LIN {X 0,Y 227.933,Z 465.716,A -85,B 0,C 180,E1 -20092.329,E2 -20092.329} C_VEL
LIN {X 0,Y 227.945,Z 465.715,A -85,B 0,C 180,E1 -20096.602,E2 -20096.602} C_VEL
LIN {X 0,Y 227.902,Z 465.721,A -85,B 0,C 180,E1 -20100.292,E2 -20100.292} C_VEL
LIN {X 0,Y 227.747,Z 465.74,A -85,B 0,C 180,E1 -20103.742,E2 -20103.742} C_VEL
LIN {X 0,Y 227.512,Z 465.771,A -85,B 0,C 180,E1 -20106.566,E2 -20106.566} C_VEL
LIN {X 0,Y 227.279,Z 465.972,A -85,B 0,C 180,E1 -20109.146,E2 -20109.146} C_VEL
LIN {X 0,Y 231.965,Z 479.924,A -85,B 0,C 180,E1 -20110.648,E2 -20110.648} C_VEL
LIN {X 0,Y 235.68,Z 494.545,A -85,B 0,C 180,E1 -20112.428,E2 -20112.428} C_VEL
LIN {X 0,Y 238.49,Z 507.946,A -85,B 0,C 180,E1 -20114.33,E2 -20114.33} C_VEL
LIN {X 0,Y 238.944,Z 511.073,A -85,B 0,C 180,E1 -20114.799,E2 -20114.799} C_VEL
LIN {X 0,Y 236.811,Z 523.709,A -85,B 0,C 180,E1 -20116.662,E2 -20116.662} C_VEL
LIN {X 0,Y 234.596,Z 535.4,A -85,B 0,C 180,E1 -20118.77,E2 -20118.77} C_VEL
LIN {X 0,Y 232.314,Z 547.285,A -85,B 0,C 180,E1 -20121.409,E2 -20121.409} C_VEL
LIN {X 0,Y 230.404,Z 556.987,A -85,B 0,C 180,E1 -20124.042,E2 -20124.042} C_VEL
LIN {X 0,Y 228.727,Z 565.771,A -85,B 0,C 180,E1 -20126.948,E2 -20126.948} C_VEL
LIN {X 0,Y 227.575,Z 572.918,A -85,B 0,C 180,E1 -20129.847,E2 -20129.847} C_VEL
LIN {X 0,Y 226.553,Z 579.643,A -85,B 0,C 180,E1 -20133.269,E2 -20133.269} C_VEL
LIN {X 0,Y 225.996,Z 584.123,A -85,B 0,C 180,E1 -20136.154,E2 -20136.154} C_VEL
LIN {X 0,Y 225.683,Z 587.632,A -85,B 0,C 180,E1 -20139.101,E2 -20139.101} C_VEL
LIN {X 0,Y 225.632,Z 589.987,A -85,B 0,C 180,E1 -20141.851,E2 -20141.851} C_VEL
LIN {X 0,Y 226.022,Z 591.964,A -85,B 0,C 180,E1 -20145.596,E2 -20145.596} C_VEL
LIN {X 0,Y 226.859,Z 592.527,A -85,B 0,C 180,E1 -20149.287,E2 -20149.287} C_VEL
LIN {X 0,Y 228.331,Z 591.732,A -85,B 0,C 180,E1 -20152.927,E2 -20152.927} C_VEL
LIN {X 0,Y 230.472,Z 589.612,A -85,B 0,C 180,E1 -20156.503,E2 -20156.503} C_VEL
LIN {X 0,Y 233.31,Z 586.131,A -85,B 0,C 180,E1 -20160,E2 -20160} C_VEL
LIN {X 0,Y 237.001,Z 581.247,A -85,B 0,C 180,E1 -20163.4,E2 -20163.4} C_VEL
LIN {X 0,Y 241.37,Z 574.833,A -85,B 0,C 180,E1 -20166.688,E2 -20166.688} C_VEL
LIN {X 0,Y 245.945,Z 567.842,A -85,B 0,C 180,E1 -20169.457,E2 -20169.457} C_VEL
LIN {X 0,Y 251.115,Z 559.281,A -85,B 0,C 180,E1 -20172.117,E2 -20172.117} C_VEL
LIN {X 0,Y 256.753,Z 549.023,A -85,B 0,C 180,E1 -20174.666,E2 -20174.666} C_VEL
LIN {X 0,Y 262.048,Z 538.351,A -85,B 0,C 180,E1 -20176.757,E2 -20176.757} C_VEL
LIN {X 0,Y 262.469,Z 536.8,A -85,B 0,C 180,E1 -20177.13,E2 -20177.13} C_VEL
LIN {X 0,Y 262.228,Z 531.504,A -85,B 0,C 180,E1 -20179.059,E2 -20179.059} C_VEL
LIN {X 0,Y 261.499,Z 526.204,A -85,B 0,C 180,E1 -20181.251,E2 -20181.251} C_VEL
LIN {X 0,Y 260.237,Z 521.055,A -85,B 0,C 180,E1 -20183.897,E2 -20183.897} C_VEL
LIN {X 0,Y 259.201,Z 518.357,A -85,B 0,C 180,E1 -20185.71,E2 -20185.71} C_VEL
LIN {X 0,Y 258.204,Z 516.399,A -85,B 0,C 180,E1 -20187.563,E2 -20187.563} C_VEL
LIN {X 0,Y 257.317,Z 514.957,A -85,B 0,C 180,E1 -20189.447,E2 -20189.447} C_VEL
LIN {X 0,Y 256.6,Z 513.704,A -85,B 0,C 180,E1 -20191.892,E2 -20191.892} C_VEL
LIN {X 0,Y 256.346,Z 513.407,A -85,B 0,C 180,E1 -20193.252,E2 -20193.252} C_VEL
LIN {X 0,Y 256.04,Z 513.801,A -85,B 0,C 180,E1 -20195.199,E2 -20195.199} C_VEL
LIN {X 0,Y 256.535,Z 515.763,A -85,B 0,C 180,E1 -20199.058,E2 -20199.058} C_VEL
LIN {X 0,Y 257.505,Z 521.048,A -85,B 0,C 180,E1 -20203.025,E2 -20203.025} C_VEL
LIN {X 0,Y 258.198,Z 524.969,A -85,B 0,C 180,E1 -20205.048,E2 -20205.048} C_VEL
LIN {X 0,Y 258.639,Z 529.116,A -85,B 0,C 180,E1 -20206.725,E2 -20206.725} C_VEL
LIN {X 0,Y 258.68,Z 537.141,A -85,B 0,C 180,E1 -20209.305,E2 -20209.305} C_VEL
LIN {X 0,Y 258.66,Z 537.501,A -85,B 0,C 180,E1 -20209.412,E2 -20209.412} C_VEL
LIN {X 0,Y 257.951,Z 541.489,A -85,B 0,C 180,E1 -20210.377,E2 -20210.377} C_VEL
LIN {X 0,Y 256.451,Z 545.94,A -85,B 0,C 180,E1 -20211.202,E2 -20211.202} C_VEL
LIN {X 0,Y 251.158,Z 557.863,A -85,B 0,C 180,E1 -20213.305,E2 -20213.305} C_VEL
LIN {X 0,Y 250.114,Z 560.562,A -85,B 0,C 180,E1 -20213.936,E2 -20213.936} C_VEL
LIN {X 0,Y 247.79,Z 566.678,A -85,B 0,C 180,E1 -20215.442,E2 -20215.442} C_VEL
LIN {X 0,Y 242.545,Z 575.941,A -85,B 0,C 180,E1 -20217.585,E2 -20217.585} C_VEL
LIN {X 0,Y 237.104,Z 585.099,A -85,B 0,C 180,E1 -20220.233,E2 -20220.233} C_VEL
LIN {X 0,Y 233.036,Z 591.862,A -85,B 0,C 180,E1 -20222.619,E2 -20222.619} C_VEL
LIN {X 0,Y 228.918,Z 598.493,A -85,B 0,C 180,E1 -20225.515,E2 -20225.515} C_VEL
LIN {X 0,Y 225.038,Z 604.726,A -85,B 0,C 180,E1 -20228.953,E2 -20228.953} C_VEL
LIN {X 0,Y 222.166,Z 609.536,A -85,B 0,C 180,E1 -20232.511,E2 -20232.511} C_VEL
LIN {X 0,Y 220.591,Z 612.29,A -85,B 0,C 180,E1 -20235.234,E2 -20235.234} C_VEL
LIN {X 0,Y 219.223,Z 614.884,A -85,B 0,C 180,E1 -20238.91,E2 -20238.91} C_VEL
LIN {X 0,Y 218.689,Z 616.234,A -85,B 0,C 180,E1 -20242.614,E2 -20242.614} C_VEL
LIN {X 0,Y 218.848,Z 616.308,A -85,B 0,C 180,E1 -20246.318,E2 -20246.318} C_VEL
LIN {X 0,Y 219.08,Z 615.033,A -85,B 0,C 180,E1 -20250,E2 -20250} C_VEL
LIN {X 0,Y 218.976,Z 612.273,A -85,B 0,C 180,E1 -20253.68,E2 -20253.68} C_VEL
LIN {X 0,Y 219.06,Z 609.777,A -85,B 0,C 180,E1 -20255.981,E2 -20255.981} C_VEL
LIN {X 0,Y 219.178,Z 605.128,A -85,B 0,C 180,E1 -20259.226,E2 -20259.226} C_VEL
LIN {X 0,Y 219.659,Z 600.055,A -85,B 0,C 180,E1 -20262.003,E2 -20262.003} C_VEL
LIN {X 0,Y 220.616,Z 592.746,A -85,B 0,C 180,E1 -20265.237,E2 -20265.237} C_VEL
LIN {X 0,Y 222.212,Z 583.656,A -85,B 0,C 180,E1 -20268.437,E2 -20268.437} C_VEL
LIN {X 0,Y 224.07,Z 574.212,A -85,B 0,C 180,E1 -20271.143,E2 -20271.143} C_VEL
LIN {X 0,Y 226.416,Z 562.842,A -85,B 0,C 180,E1 -20273.798,E2 -20273.798} C_VEL
LIN {X 0,Y 228.937,Z 550.545,A -85,B 0,C 180,E1 -20276.121,E2 -20276.121} C_VEL
LIN {X 0,Y 228.849,Z 545.123,A -85,B 0,C 180,E1 -20277.052,E2 -20277.052} C_VEL
LIN {X 0,Y 227.742,Z 532.027,A -85,B 0,C 180,E1 -20279.08,E2 -20279.08} C_VEL
LIN {X 0,Y 226.226,Z 517.932,A -85,B 0,C 180,E1 -20280.909,E2 -20280.909} C_VEL
LIN {X 0,Y 224.184,Z 502.881,A -85,B 0,C 180,E1 -20282.529,E2 -20282.529} C_VEL
LIN {X 0,Y 221.762,Z 487.259,A -85,B 0,C 180,E1 -20283.908,E2 -20283.908} C_VEL
LIN {X 0,Y 222.836,Z 482.859,A -85,B 0,C 180,E1 -20287.957,E2 -20287.957} C_VEL
LIN {X 0,Y 223.128,Z 479.233,A -85,B 0,C 180,E1 -20291.41,E2 -20291.41} C_VEL
LIN {X 0,Y 222.752,Z 476.696,A -85,B 0,C 180,E1 -20293.956,E2 -20293.956} C_VEL
LIN {X 0,Y 221.937,Z 472.506,A -85,B 0,C 180,E1 -20298.318,E2 -20298.318} C_VEL
LIN {X 0,Y 221.216,Z 468.39,A -85,B 0,C 180,E1 -20302.87,E2 -20302.87} C_VEL
LIN {X 0,Y 220.928,Z 466.591,A -85,B 0,C 180,E1 -20305.068,E2 -20305.068} C_VEL
LIN {X 0,Y 220.865,Z 466.599,A -85,B 0,C 180,E1 -20309.395,E2 -20309.395} C_VEL
LIN {X 0,Y 220.892,Z 466.589,A -85,B 0,C 180,E1 -20313.549,E2 -20313.549} C_VEL
LIN {X 0,Y 220.875,Z 466.595,A -85,B 0,C 180,E1 -20317.553,E2 -20317.553} C_VEL
LIN {X 0,Y 220.981,Z 466.583,A -85,B 0,C 180,E1 -20322.571,E2 -20322.571} C_VEL
LIN {X 0,Y 221.023,Z 466.578,A -85,B 0,C 180,E1 -20327.14,E2 -20327.14} C_VEL
LIN {X 0,Y 221.233,Z 466.551,A -85,B 0,C 180,E1 -20330.861,E2 -20330.861} C_VEL
LIN {X 0,Y 221.286,Z 466.543,A -85,B 0,C 180,E1 -20332.702,E2 -20332.702} C_VEL
LIN {X 0,Y 221.51,Z 466.517,A -85,B 0,C 180,E1 -20338.182,E2 -20338.182} C_VEL
LIN {X 0,Y 221.512,Z 466.512,A -85,B 0,C 180,E1 -20341.819,E2 -20341.819} C_VEL
LIN {X 0,Y 221.288,Z 466.543,A -85,B 0,C 180,E1 -20347.299,E2 -20347.299} C_VEL
LIN {X 0,Y 221.109,Z 466.564,A -85,B 0,C 180,E1 -20350.995,E2 -20350.995} C_VEL
LIN {X 0,Y 221.014,Z 466.579,A -85,B 0,C 180,E1 -20356.63,E2 -20356.63} C_VEL
LIN {X 0,Y 220.89,Z 466.594,A -85,B 0,C 180,E1 -20360.487,E2 -20360.487} C_VEL
LIN {X 0,Y 220.865,Z 466.599,A -85,B 0,C 180,E1 -20364.436,E2 -20364.436} C_VEL
LIN {X 0,Y 220.835,Z 466.599,A -85,B 0,C 180,E1 -20368.514,E2 -20368.514} C_VEL
LIN {X 0,Y 220.822,Z 466.602,A -85,B 0,C 180,E1 -20372.756,E2 -20372.756} C_VEL
LIN {X 0,Y 220.838,Z 466.596,A -85,B 0,C 180,E1 -20377.289,E2 -20377.289} C_VEL
LIN {X 0,Y 220.769,Z 466.612,A -85,B 0,C 180,E1 -20381.953,E2 -20381.953} C_VEL
LIN {X 0,Y 220.802,Z 466.603,A -85,B 0,C 180,E1 -20385.554,E2 -20385.554} C_VEL
LIN {X 0,Y 220.806,Z 466.606,A -85,B 0,C 180,E1 -20389.809,E2 -20389.809} C_VEL
LIN {X 0,Y 220.835,Z 466.599,A -85,B 0,C 180,E1 -20392.796,E2 -20392.796} C_VEL
LIN {X 0,Y 220.826,Z 466.601,A -85,B 0,C 180,E1 -20397.246,E2 -20397.246} C_VEL
LIN {X 0,Y 220.84,Z 466.601,A -85,B 0,C 180,E1 -20401.488,E2 -20401.488} C_VEL
LIN {X 0,Y 220.87,Z 466.596,A -85,B 0,C 180,E1 -20405.566,E2 -20405.566} C_VEL
LIN {X 0,Y 220.895,Z 466.595,A -85,B 0,C 180,E1 -20409.515,E2 -20409.515} C_VEL
LIN {X 0,Y 221.02,Z 466.576,A -85,B 0,C 180,E1 -20413.371,E2 -20413.371} C_VEL
LIN {X 0,Y 221.015,Z 466.579,A -85,B 0,C 180,E1 -20417.139,E2 -20417.139} C_VEL
LIN {X 0,Y 221.201,Z 466.552,A -85,B 0,C 180,E1 -20420.859,E2 -20420.859} C_VEL
LIN {X 0,Y 221.133,Z 466.563,A -85,B 0,C 180,E1 -20424.529,E2 -20424.529} C_VEL
LIN {X 0,Y 221.515,Z 466.514,A -85,B 0,C 180,E1 -20428.182,E2 -20428.182} C_VEL
LIN {X 0,Y 221.516,Z 466.516,A -85,B 0,C 180,E1 -20431.818,E2 -20431.818} C_VEL
LIN {X 0,Y 221.275,Z 466.546,A -85,B 0,C 180,E1 -20437.299,E2 -20437.299} C_VEL
LIN {X 0,Y 221.085,Z 466.567,A -85,B 0,C 180,E1 -20440.995,E2 -20440.995} C_VEL
LIN {X 0,Y 221.02,Z 466.578,A -85,B 0,C 180,E1 -20446.629,E2 -20446.629} C_VEL
LIN {X 0,Y 220.895,Z 466.594,A -85,B 0,C 180,E1 -20450.485,E2 -20450.485} C_VEL
LIN {X 0,Y 220.87,Z 466.596,A -85,B 0,C 180,E1 -20454.434,E2 -20454.434} C_VEL
LIN {X 0,Y 220.837,Z 466.602,A -85,B 0,C 180,E1 -20458.513,E2 -20458.513} C_VEL
LIN {X 0,Y 220.738,Z 466.616,A -85,B 0,C 180,E1 -20462.769,E2 -20462.769} C_VEL
LIN {X 0,Y 220.375,Z 466.661,A -85,B 0,C 180,E1 -20467.128,E2 -20467.128} C_VEL
LIN {X 0,Y 220.266,Z 466.673,A -85,B 0,C 180,E1 -20468.475,E2 -20468.475} C_VEL
LIN {X 0,Y 225.146,Z 481.341,A -85,B 0,C 180,E1 -20470.14,E2 -20470.14} C_VEL
LIN {X 0,Y 228.581,Z 494.783,A -85,B 0,C 180,E1 -20471.857,E2 -20471.857} C_VEL
LIN {X 0,Y 231.312,Z 507.592,A -85,B 0,C 180,E1 -20473.725,E2 -20473.725} C_VEL
LIN {X 0,Y 232.051,Z 511.762,A -85,B 0,C 180,E1 -20474.38,E2 -20474.38} C_VEL
LIN {X 0,Y 229.637,Z 525.37,A -85,B 0,C 180,E1 -20476.479,E2 -20476.479} C_VEL
LIN {X 0,Y 227.197,Z 538.03,A -85,B 0,C 180,E1 -20478.902,E2 -20478.902} C_VEL
LIN {X 0,Y 225.143,Z 548.537,A -85,B 0,C 180,E1 -20481.368,E2 -20481.368} C_VEL
LIN {X 0,Y 223.312,Z 557.476,A -85,B 0,C 180,E1 -20483.892,E2 -20483.892} C_VEL
LIN {X 0,Y 221.652,Z 566.13,A -85,B 0,C 180,E1 -20486.841,E2 -20486.841} C_VEL
LIN {X 0,Y 220.449,Z 573.357,A -85,B 0,C 180,E1 -20489.859,E2 -20489.859} C_VEL
LIN {X 0,Y 219.422,Z 580.028,A -85,B 0,C 180,E1 -20493.358,E2 -20493.358} C_VEL
LIN {X 0,Y 218.87,Z 584.506,A -85,B 0,C 180,E1 -20496.335,E2 -20496.335} C_VEL
LIN {X 0,Y 218.598,Z 587.919,A -85,B 0,C 180,E1 -20499.289,E2 -20499.289} C_VEL
LIN {X 0,Y 218.619,Z 591.077,A -85,B 0,C 180,E1 -20503.182,E2 -20503.182} C_VEL
LIN {X 0,Y 218.886,Z 592.073,A -85,B 0,C 180,E1 -20505.116,E2 -20505.116} C_VEL
LIN {X 0,Y 219.664,Z 593.005,A -85,B 0,C 180,E1 -20508.932,E2 -20508.932} C_VEL
LIN {X 0,Y 221.117,Z 592.584,A -85,B 0,C 180,E1 -20512.695,E2 -20512.695} C_VEL
LIN {X 0,Y 223.243,Z 590.848,A -85,B 0,C 180,E1 -20516.39,E2 -20516.39} C_VEL
LIN {X 0,Y 226.139,Z 587.824,A -85,B 0,C 180,E1 -20520,E2 -20520} C_VEL
LIN {X 0,Y 229.886,Z 583.396,A -85,B 0,C 180,E1 -20523.505,E2 -20523.505} C_VEL
LIN {X 0,Y 234.377,Z 577.554,A -85,B 0,C 180,E1 -20526.889,E2 -20526.889} C_VEL
LIN {X 0,Y 239.04,Z 571.047,A -85,B 0,C 180,E1 -20529.733,E2 -20529.733} C_VEL
LIN {X 0,Y 244.347,Z 563.122,A -85,B 0,C 180,E1 -20532.458,E2 -20532.458} C_VEL
LIN {X 0,Y 250.086,Z 553.566,A -85,B 0,C 180,E1 -20535.067,E2 -20535.067} C_VEL
LIN {X 0,Y 256.512,Z 541.921,A -85,B 0,C 180,E1 -20537.54,E2 -20537.54} C_VEL
LIN {X 0,Y 257.217,Z 540.45,A -85,B 0,C 180,E1 -20537.846,E2 -20537.846} C_VEL
LIN {X 0,Y 257.174,Z 534.976,A -85,B 0,C 180,E1 -20539.975,E2 -20539.975} C_VEL
LIN {X 0,Y 256.547,Z 529.42,A -85,B 0,C 180,E1 -20542.552,E2 -20542.552} C_VEL
LIN {X 0,Y 255.656,Z 525.566,A -85,B 0,C 180,E1 -20544.885,E2 -20544.885} C_VEL
LIN {X 0,Y 255.128,Z 523.925,A -85,B 0,C 180,E1 -20546.152,E2 -20546.152} C_VEL
LIN {X 0,Y 254.284,Z 522.111,A -85,B 0,C 180,E1 -20548.025,E2 -20548.025} C_VEL
LIN {X 0,Y 253.153,Z 519.909,A -85,B 0,C 180,E1 -20551.835,E2 -20551.835} C_VEL
LIN {X 0,Y 252.828,Z 519.72,A -85,B 0,C 180,E1 -20553.776,E2 -20553.776} C_VEL
LIN {X 0,Y 252.749,Z 521.142,A -85,B 0,C 180,E1 -20557.715,E2 -20557.715} C_VEL
LIN {X 0,Y 253.007,Z 521.98,A -85,B 0,C 180,E1 -20558.944,E2 -20558.944} C_VEL
LIN {X 0,Y 253.742,Z 527.686,A -85,B 0,C 180,E1 -20563.188,E2 -20563.188} C_VEL
LIN {X 0,Y 254.15,Z 532.263,A -85,B 0,C 180,E1 -20565.453,E2 -20565.453} C_VEL
LIN {X 0,Y 254.1,Z 537.129,A -85,B 0,C 180,E1 -20567.247,E2 -20567.247} C_VEL
LIN {X 0,Y 253.519,Z 544.054,A -85,B 0,C 180,E1 -20569.445,E2 -20569.445} C_VEL
LIN {X 0,Y 252.27,Z 551.866,A -85,B 0,C 180,E1 -20571.658,E2 -20571.658} C_VEL
LIN {X 0,Y 250.114,Z 560.562,A -85,B 0,C 180,E1 -20573.936,E2 -20573.936} C_VEL
LIN {X 0,Y 248.605,Z 563.369,A -85,B 0,C 180,E1 -20574.482,E2 -20574.482} C_VEL
LIN {X 0,Y 244.498,Z 568.109,A -85,B 0,C 180,E1 -20575.042,E2 -20575.042} C_VEL
LIN {X 0,Y 240.024,Z 572.728,A -85,B 0,C 180,E1 -20575.59,E2 -20575.59} C_VEL
LIN {X 0,Y 237.983,Z 575.357,A -85,B 0,C 180,E1 -20576.133,E2 -20576.133} C_VEL
LIN {X 0,Y 231.714,Z 585.092,A -85,B 0,C 180,E1 -20578.962,E2 -20578.962} C_VEL
LIN {X 0,Y 227.435,Z 591.666,A -85,B 0,C 180,E1 -20581.383,E2 -20581.383} C_VEL
LIN {X 0,Y 222.486,Z 599.066,A -85,B 0,C 180,E1 -20584.758,E2 -20584.758} C_VEL
LIN {X 0,Y 218.395,Z 604.989,A -85,B 0,C 180,E1 -20588.28,E2 -20588.28} C_VEL
LIN {X 0,Y 216.035,Z 608.6,A -85,B 0,C 180,E1 -20591.016,E2 -20591.016} C_VEL
LIN {X 0,Y 213.687,Z 612.238,A -85,B 0,C 180,E1 -20594.745,E2 -20594.745} C_VEL
LIN {X 0,Y 212.221,Z 614.651,A -85,B 0,C 180,E1 -20598.539,E2 -20598.539} C_VEL
LIN {X 0,Y 211.617,Z 615.826,A -85,B 0,C 180,E1 -20602.366,E2 -20602.366} C_VEL
LIN {X 0,Y 211.782,Z 615.748,A -85,B 0,C 180,E1 -20606.195,E2 -20606.195} C_VEL
LIN {X 0,Y 212.008,Z 614.315,A -85,B 0,C 180,E1 -20610,E2 -20610} C_VEL
LIN {X 0,Y 211.921,Z 611.397,A -85,B 0,C 180,E1 -20613.803,E2 -20613.803} C_VEL
LIN {X 0,Y 211.995,Z 608.149,A -85,B 0,C 180,E1 -20616.662,E2 -20616.662} C_VEL
LIN {X 0,Y 212.278,Z 602.371,A -85,B 0,C 180,E1 -20620.491,E2 -20620.491} C_VEL
LIN {X 0,Y 213.095,Z 595.764,A -85,B 0,C 180,E1 -20623.834,E2 -20623.834} C_VEL
LIN {X 0,Y 214.344,Z 587.466,A -85,B 0,C 180,E1 -20627.163,E2 -20627.163} C_VEL
LIN {X 0,Y 216.03,Z 578.874,A -85,B 0,C 180,E1 -20629.973,E2 -20629.973} C_VEL
LIN {X 0,Y 218.126,Z 568.537,A -85,B 0,C 180,E1 -20632.745,E2 -20632.745} C_VEL
LIN {X 0,Y 220.555,Z 557.18,A -85,B 0,C 180,E1 -20635.226,E2 -20635.226} C_VEL
LIN {X 0,Y 222.085,Z 549.546,A -85,B 0,C 180,E1 -20636.64,E2 -20636.64} C_VEL
LIN {X 0,Y 221.171,Z 537.512,A -85,B 0,C 180,E1 -20638.709,E2 -20638.709} C_VEL
LIN {X 0,Y 219.89,Z 523.377,A -85,B 0,C 180,E1 -20640.755,E2 -20640.755} C_VEL
LIN {X 0,Y 218.104,Z 508.822,A -85,B 0,C 180,E1 -20642.525,E2 -20642.525} C_VEL
LIN {X 0,Y 215.835,Z 493.244,A -85,B 0,C 180,E1 -20644.062,E2 -20644.062} C_VEL
LIN {X 0,Y 214.841,Z 486.84,A -85,B 0,C 180,E1 -20644.654,E2 -20644.654} C_VEL
LIN {X 0,Y 215.845,Z 482.72,A -85,B 0,C 180,E1 -20648.607,E2 -20648.607} C_VEL
LIN {X 0,Y 216.04,Z 479.739,A -85,B 0,C 180,E1 -20651.565,E2 -20651.565} C_VEL
LIN {X 0,Y 215.354,Z 475.599,A -85,B 0,C 180,E1 -20655.885,E2 -20655.885} C_VEL
LIN {X 0,Y 214.541,Z 471.596,A -85,B 0,C 180,E1 -20660.299,E2 -20660.299} C_VEL
LIN {X 0,Y 213.893,Z 467.466,A -85,B 0,C 180,E1 -20665.171,E2 -20665.171} C_VEL
LIN {X 0,Y 213.778,Z 467.481,A -85,B 0,C 180,E1 -20670.454,E2 -20670.454} C_VEL
LIN {X 0,Y 213.799,Z 467.473,A -85,B 0,C 180,E1 -20674.702,E2 -20674.702} C_VEL
LIN {X 0,Y 213.81,Z 467.478,A -85,B 0,C 180,E1 -20678.803,E2 -20678.803} C_VEL
LIN {X 0,Y 213.941,Z 467.459,A -85,B 0,C 180,E1 -20682.804,E2 -20682.804} C_VEL
LIN {X 0,Y 213.977,Z 467.456,A -85,B 0,C 180,E1 -20686.708,E2 -20686.708} C_VEL
LIN {X 0,Y 214.165,Z 467.433,A -85,B 0,C 180,E1 -20690.557,E2 -20690.557} C_VEL
LIN {X 0,Y 214.224,Z 467.424,A -85,B 0,C 180,E1 -20692.46,E2 -20692.46} C_VEL
LIN {X 0,Y 214.443,Z 467.397,A -85,B 0,C 180,E1 -20698.122,E2 -20698.122} C_VEL
LIN {X 0,Y 214.547,Z 467.383,A -85,B 0,C 180,E1 -20700,E2 -20700} C_VEL
LIN {X 0,Y 214.445,Z 467.392,A -85,B 0,C 180,E1 -20701.878,E2 -20701.878} C_VEL
LIN {X 0,Y 214.226,Z 467.423,A -85,B 0,C 180,E1 -20707.541,E2 -20707.541} C_VEL
LIN {X 0,Y 214.042,Z 467.443,A -85,B 0,C 180,E1 -20711.362,E2 -20711.362} C_VEL
LIN {X 0,Y 213.929,Z 467.46,A -85,B 0,C 180,E1 -20715.238,E2 -20715.238} C_VEL
LIN {X 0,Y 213.837,Z 467.468,A -85,B 0,C 180,E1 -20719.188,E2 -20719.188} C_VEL
LIN {X 0,Y 213.846,Z 467.471,A -85,B 0,C 180,E1 -20723.228,E2 -20723.228} C_VEL
LIN {X 0,Y 213.828,Z 467.47,A -85,B 0,C 180,E1 -20727.451,E2 -20727.451} C_VEL
LIN {X 0,Y 213.778,Z 467.48,A -85,B 0,C 180,E1 -20731.736,E2 -20731.736} C_VEL
LIN {X 0,Y 213.747,Z 467.481,A -85,B 0,C 180,E1 -20736.288,E2 -20736.288} C_VEL
LIN {X 0,Y 213.711,Z 467.487,A -85,B 0,C 180,E1 -20741.126,E2 -20741.126} C_VEL
LIN {X 0,Y 213.748,Z 467.482,A -85,B 0,C 180,E1 -20746.333,E2 -20746.333} C_VEL
LIN {X 0,Y 213.74,Z 467.484,A -85,B 0,C 180,E1 -20749.137,E2 -20749.137} C_VEL
LIN {X 0,Y 213.755,Z 467.483,A -85,B 0,C 180,E1 -20753.715,E2 -20753.715} C_VEL
LIN {X 0,Y 213.798,Z 467.477,A -85,B 0,C 180,E1 -20758.725,E2 -20758.725} C_VEL
LIN {X 0,Y 213.828,Z 467.47,A -85,B 0,C 180,E1 -20762.604,E2 -20762.604} C_VEL
LIN {X 0,Y 213.855,Z 467.47,A -85,B 0,C 180,E1 -20766.953,E2 -20766.953} C_VEL
LIN {X 0,Y 213.947,Z 467.455,A -85,B 0,C 180,E1 -20772.804,E2 -20772.804} C_VEL
LIN {X 0,Y 213.956,Z 467.457,A -85,B 0,C 180,E1 -20776.707,E2 -20776.707} C_VEL
LIN {X 0,Y 214.139,Z 467.431,A -85,B 0,C 180,E1 -20780.555,E2 -20780.555} C_VEL
LIN {X 0,Y 214.094,Z 467.44,A -85,B 0,C 180,E1 -20784.348,E2 -20784.348} C_VEL
LIN {X 0,Y 214.448,Z 467.394,A -85,B 0,C 180,E1 -20788.122,E2 -20788.122} C_VEL
LIN {X 0,Y 214.554,Z 467.38,A -85,B 0,C 180,E1 -20790,E2 -20790} C_VEL
LIN {X 0,Y 214.449,Z 467.396,A -85,B 0,C 180,E1 -20791.878,E2 -20791.878} C_VEL
LIN {X 0,Y 214.212,Z 467.424,A -85,B 0,C 180,E1 -20797.541,E2 -20797.541} C_VEL
LIN {X 0,Y 214.011,Z 467.451,A -85,B 0,C 180,E1 -20801.364,E2 -20801.364} C_VEL
LIN {X 0,Y 213.938,Z 467.463,A -85,B 0,C 180,E1 -20805.236,E2 -20805.236} C_VEL
LIN {X 0,Y 213.871,Z 467.47,A -85,B 0,C 180,E1 -20809.184,E2 -20809.184} C_VEL
LIN {X 0,Y 213.85,Z 467.472,A -85,B 0,C 180,E1 -20813.226,E2 -20813.226} C_VEL
LIN {X 0,Y 213.831,Z 467.475,A -85,B 0,C 180,E1 -20817.449,E2 -20817.449} C_VEL
LIN {X 0,Y 213.702,Z 467.49,A -85,B 0,C 180,E1 -20821.748,E2 -20821.748} C_VEL
LIN {X 0,Y 213.58,Z 467.507,A -85,B 0,C 180,E1 -20824.649,E2 -20824.649} C_VEL
LIN {X 0,Y 213.276,Z 467.543,A -85,B 0,C 180,E1 -20827.787,E2 -20827.787} C_VEL
LIN {X 0,Y 218.596,Z 483.564,A -85,B 0,C 180,E1 -20829.716,E2 -20829.716} C_VEL
LIN {X 0,Y 222.143,Z 497.665,A -85,B 0,C 180,E1 -20831.634,E2 -20831.634} C_VEL
LIN {X 0,Y 224.936,Z 511.345,A -85,B 0,C 180,E1 -20833.762,E2 -20833.762} C_VEL
LIN {X 0,Y 225.026,Z 513.326,A -85,B 0,C 180,E1 -20834.082,E2 -20834.082} C_VEL
LIN {X 0,Y 222.561,Z 526.773,A -85,B 0,C 180,E1 -20836.25,E2 -20836.25} C_VEL
LIN {X 0,Y 220.249,Z 538.308,A -85,B 0,C 180,E1 -20838.538,E2 -20838.538} C_VEL
LIN {X 0,Y 218.106,Z 548.939,A -85,B 0,C 180,E1 -20841.103,E2 -20841.103} C_VEL
LIN {X 0,Y 215.946,Z 559.211,A -85,B 0,C 180,E1 -20844.139,E2 -20844.139} C_VEL
LIN {X 0,Y 214.322,Z 567.718,A -85,B 0,C 180,E1 -20847.243,E2 -20847.243} C_VEL
LIN {X 0,Y 213.01,Z 575.729,A -85,B 0,C 180,E1 -20850.878,E2 -20850.878} C_VEL
LIN {X 0,Y 212.104,Z 581.978,A -85,B 0,C 180,E1 -20854.484,E2 -20854.484} C_VEL
LIN {X 0,Y 211.645,Z 586.094,A -85,B 0,C 180,E1 -20857.551,E2 -20857.551} C_VEL
LIN {X 0,Y 211.434,Z 589.234,A -85,B 0,C 180,E1 -20860.585,E2 -20860.585} C_VEL
LIN {X 0,Y 211.719,Z 592.018,A -85,B 0,C 180,E1 -20864.599,E2 -20864.599} C_VEL
LIN {X 0,Y 212.465,Z 593.367,A -85,B 0,C 180,E1 -20868.552,E2 -20868.552} C_VEL
LIN {X 0,Y 213.88,Z 593.355,A -85,B 0,C 180,E1 -20872.447,E2 -20872.447} C_VEL
LIN {X 0,Y 216.038,Z 592.042,A -85,B 0,C 180,E1 -20876.269,E2 -20876.269} C_VEL
LIN {X 0,Y 218.969,Z 589.433,A -85,B 0,C 180,E1 -20880,E2 -20880} C_VEL
LIN {X 0,Y 222.796,Z 585.477,A -85,B 0,C 180,E1 -20883.617,E2 -20883.617} C_VEL
LIN {X 0,Y 227.345,Z 580.102,A -85,B 0,C 180,E1 -20887.103,E2 -20887.103} C_VEL
LIN {X 0,Y 232.863,Z 573.123,A -85,B 0,C 180,E1 -20890.433,E2 -20890.433} C_VEL
LIN {X 0,Y 238.131,Z 565.875,A -85,B 0,C 180,E1 -20893.115,E2 -20893.115} C_VEL
LIN {X 0,Y 244.374,Z 556.487,A -85,B 0,C 180,E1 -20895.855,E2 -20895.855} C_VEL
LIN {X 0,Y 250.026,Z 547.164,A -85,B 0,C 180,E1 -20898.011,E2 -20898.011} C_VEL
LIN {X 0,Y 251.959,Z 543.679,A -85,B 0,C 180,E1 -20898.71,E2 -20898.71} C_VEL
LIN {X 0,Y 252.189,Z 539.702,A -85,B 0,C 180,E1 -20900.387,E2 -20900.387} C_VEL
LIN {X 0,Y 251.94,Z 534.443,A -85,B 0,C 180,E1 -20902.995,E2 -20902.995} C_VEL
LIN {X 0,Y 251.47,Z 531.582,A -85,B 0,C 180,E1 -20904.785,E2 -20904.785} C_VEL
LIN {X 0,Y 250.87,Z 529.361,A -85,B 0,C 180,E1 -20906.63,E2 -20906.63} C_VEL
LIN {X 0,Y 249.916,Z 527.232,A -85,B 0,C 180,E1 -20909.338,E2 -20909.338} C_VEL
LIN {X 0,Y 249.334,Z 525.857,A -85,B 0,C 180,E1 -20912.381,E2 -20912.381} C_VEL
LIN {X 0,Y 248.967,Z 526.133,A -85,B 0,C 180,E1 -20915.054,E2 -20915.054} C_VEL
LIN {X 0,Y 249.172,Z 527.665,A -85,B 0,C 180,E1 -20918.354,E2 -20918.354} C_VEL
LIN {X 0,Y 249.324,Z 531.222,A -85,B 0,C 180,E1 -20921.374,E2 -20921.374} C_VEL
LIN {X 0,Y 249.632,Z 533.441,A -85,B 0,C 180,E1 -20922.948,E2 -20922.948} C_VEL
LIN {X 0,Y 249.703,Z 538.15,A -85,B 0,C 180,E1 -20925.282,E2 -20925.282} C_VEL
LIN {X 0,Y 249.119,Z 543.876,A -85,B 0,C 180,E1 -20927.385,E2 -20927.385} C_VEL
LIN {X 0,Y 247.838,Z 551.375,A -85,B 0,C 180,E1 -20929.773,E2 -20929.773} C_VEL
LIN {X 0,Y 245.785,Z 559.349,A -85,B 0,C 180,E1 -20932.065,E2 -20932.065} C_VEL
LIN {X 0,Y 243.183,Z 566.556,A -85,B 0,C 180,E1 -20934.018,E2 -20934.018} C_VEL
LIN {X 0,Y 239.412,Z 573.063,A -85,B 0,C 180,E1 -20935.556,E2 -20935.556} C_VEL
LIN {X 0,Y 237.983,Z 575.357,A -85,B 0,C 180,E1 -20936.133,E2 -20936.133} C_VEL
LIN {X 0,Y 235.199,Z 579.135,A -85,B 0,C 180,E1 -20937.03,E2 -20937.03} C_VEL
LIN {X 0,Y 229.197,Z 585.083,A -85,B 0,C 180,E1 -20938.326,E2 -20938.326} C_VEL
LIN {X 0,Y 223.281,Z 590.537,A -85,B 0,C 180,E1 -20939.77,E2 -20939.77} C_VEL
LIN {X 0,Y 220.681,Z 593.435,A -85,B 0,C 180,E1 -20940.888,E2 -20940.888} C_VEL
LIN {X 0,Y 216.088,Z 599.631,A -85,B 0,C 180,E1 -20943.956,E2 -20943.956} C_VEL
LIN {X 0,Y 211.809,Z 605.321,A -85,B 0,C 180,E1 -20947.569,E2 -20947.569} C_VEL
LIN {X 0,Y 209.295,Z 608.7,A -85,B 0,C 180,E1 -20950.38,E2 -20950.38} C_VEL
LIN {X 0,Y 206.806,Z 612.144,A -85,B 0,C 180,E1 -20954.225,E2 -20954.225} C_VEL
LIN {X 0,Y 205.216,Z 614.365,A -85,B 0,C 180,E1 -20958.143,E2 -20958.143} C_VEL
LIN {X 0,Y 204.567,Z 615.376,A -85,B 0,C 180,E1 -20962.101,E2 -20962.101} C_VEL
LIN {X 0,Y 204.715,Z 615.139,A -85,B 0,C 180,E1 -20966.063,E2 -20966.063} C_VEL
LIN {X 0,Y 204.94,Z 613.552,A -85,B 0,C 180,E1 -20970,E2 -20970} C_VEL
LIN {X 0,Y 204.87,Z 610.438,A -85,B 0,C 180,E1 -20973.934,E2 -20973.934} C_VEL
LIN {X 0,Y 204.94,Z 607.092,A -85,B 0,C 180,E1 -20976.892,E2 -20976.892} C_VEL
LIN {X 0,Y 205.124,Z 602.723,A -85,B 0,C 180,E1 -20979.864,E2 -20979.864} C_VEL
LIN {X 0,Y 205.877,Z 596.371,A -85,B 0,C 180,E1 -20983.322,E2 -20983.322} C_VEL
LIN {X 0,Y 207.05,Z 588.418,A -85,B 0,C 180,E1 -20986.769,E2 -20986.769} C_VEL
LIN {X 0,Y 208.695,Z 580.148,A -85,B 0,C 180,E1 -20989.679,E2 -20989.679} C_VEL
LIN {X 0,Y 210.753,Z 570.194,A -85,B 0,C 180,E1 -20992.55,E2 -20992.55} C_VEL
LIN {X 0,Y 213.367,Z 558.095,A -85,B 0,C 180,E1 -20995.353,E2 -20995.353} C_VEL
LIN {X 0,Y 215.053,Z 549.82,A -85,B 0,C 180,E1 -20996.964,E2 -20996.964} C_VEL
LIN {X 0,Y 214.14,Z 536.908,A -85,B 0,C 180,E1 -20999.268,E2 -20999.268} C_VEL
LIN {X 0,Y 212.829,Z 522.639,A -85,B 0,C 180,E1 -21001.411,E2 -21001.411} C_VEL
LIN {X 0,Y 210.984,Z 507.337,A -85,B 0,C 180,E1 -21003.31,E2 -21003.31} C_VEL
LIN {X 0,Y 208.69,Z 492.02,A -85,B 0,C 180,E1 -21004.841,E2 -21004.841} C_VEL
LIN {X 0,Y 207.936,Z 486.54,A -85,B 0,C 180,E1 -21005.319,E2 -21005.319} C_VEL
LIN {X 0,Y 208.857,Z 482.553,A -85,B 0,C 180,E1 -21009.291,E2 -21009.291} C_VEL
LIN {X 0,Y 208.861,Z 479.661,A -85,B 0,C 180,E1 -21012.297,E2 -21012.297} C_VEL
LIN {X 0,Y 208.224,Z 475.98,A -85,B 0,C 180,E1 -21016.299,E2 -21016.299} C_VEL
LIN {X 0,Y 207.348,Z 471.697,A -85,B 0,C 180,E1 -21021.221,E2 -21021.221} C_VEL
LIN {X 0,Y 206.827,Z 468.345,A -85,B 0,C 180,E1 -21025.308,E2 -21025.308} C_VEL
LIN {X 0,Y 206.722,Z 468.361,A -85,B 0,C 180,E1 -21029.339,E2 -21029.339} C_VEL
LIN {X 0,Y 206.73,Z 468.352,A -85,B 0,C 180,E1 -21033.772,E2 -21033.772} C_VEL
LIN {X 0,Y 206.755,Z 468.353,A -85,B 0,C 180,E1 -21038.043,E2 -21038.043} C_VEL
LIN {X 0,Y 206.873,Z 468.339,A -85,B 0,C 180,E1 -21042.197,E2 -21042.197} C_VEL
LIN {X 0,Y 206.911,Z 468.333,A -85,B 0,C 180,E1 -21046.246,E2 -21046.246} C_VEL
LIN {X 0,Y 207.103,Z 468.311,A -85,B 0,C 180,E1 -21050.231,E2 -21050.231} C_VEL
LIN {X 0,Y 207.165,Z 468.302,A -85,B 0,C 180,E1 -21052.201,E2 -21052.201} C_VEL
LIN {X 0,Y 207.38,Z 468.277,A -85,B 0,C 180,E1 -21058.058,E2 -21058.058} C_VEL
LIN {X 0,Y 207.512,Z 468.259,A -85,B 0,C 180,E1 -21060,E2 -21060} C_VEL
LIN {X 0,Y 207.382,Z 468.272,A -85,B 0,C 180,E1 -21061.942,E2 -21061.942} C_VEL
LIN {X 0,Y 207.166,Z 468.303,A -85,B 0,C 180,E1 -21067.799,E2 -21067.799} C_VEL
LIN {X 0,Y 206.979,Z 468.323,A -85,B 0,C 180,E1 -21071.756,E2 -21071.756} C_VEL
LIN {X 0,Y 206.863,Z 468.341,A -85,B 0,C 180,E1 -21075.771,E2 -21075.771} C_VEL
LIN {X 0,Y 206.781,Z 468.347,A -85,B 0,C 180,E1 -21079.87,E2 -21079.87} C_VEL
LIN {X 0,Y 206.762,Z 468.355,A -85,B 0,C 180,E1 -21084.073,E2 -21084.073} C_VEL
LIN {X 0,Y 206.743,Z 468.354,A -85,B 0,C 180,E1 -21088.419,E2 -21088.419} C_VEL
LIN {X 0,Y 206.707,Z 468.36,A -85,B 0,C 180,E1 -21092.957,E2 -21092.957} C_VEL
LIN {X 0,Y 206.721,Z 468.357,A -85,B 0,C 180,E1 -21095.321,E2 -21095.321} C_VEL
LIN {X 0,Y 206.663,Z 468.368,A -85,B 0,C 180,E1 -21100.252,E2 -21100.252} C_VEL
LIN {X 0,Y 206.659,Z 468.364,A -85,B 0,C 180,E1 -21105.575,E2 -21105.575} C_VEL
LIN {X 0,Y 206.679,Z 468.366,A -85,B 0,C 180,E1 -21109.754,E2 -21109.754} C_VEL
LIN {X 0,Y 206.733,Z 468.353,A -85,B 0,C 180,E1 -21114.696,E2 -21114.696} C_VEL
LIN {X 0,Y 206.726,Z 468.359,A -85,B 0,C 180,E1 -21119.34,E2 -21119.34} C_VEL
LIN {X 0,Y 206.735,Z 468.355,A -85,B 0,C 180,E1 -21123.773,E2 -21123.773} C_VEL
LIN {X 0,Y 206.76,Z 468.355,A -85,B 0,C 180,E1 -21128.044,E2 -21128.044} C_VEL
LIN {X 0,Y 206.876,Z 468.336,A -85,B 0,C 180,E1 -21132.197,E2 -21132.197} C_VEL
LIN {X 0,Y 206.899,Z 468.336,A -85,B 0,C 180,E1 -21136.245,E2 -21136.245} C_VEL
LIN {X 0,Y 207.083,Z 468.31,A -85,B 0,C 180,E1 -21140.23,E2 -21140.23} C_VEL
LIN {X 0,Y 207.056,Z 468.317,A -85,B 0,C 180,E1 -21144.156,E2 -21144.156} C_VEL
LIN {X 0,Y 207.384,Z 468.274,A -85,B 0,C 180,E1 -21148.058,E2 -21148.058} C_VEL
LIN {X 0,Y 207.519,Z 468.256,A -85,B 0,C 180,E1 -21150,E2 -21150} C_VEL
LIN {X 0,Y 207.386,Z 468.275,A -85,B 0,C 180,E1 -21151.942,E2 -21151.942} C_VEL
LIN {X 0,Y 207.152,Z 468.302,A -85,B 0,C 180,E1 -21157.799,E2 -21157.799} C_VEL
LIN {X 0,Y 206.935,Z 468.332,A -85,B 0,C 180,E1 -21161.758,E2 -21161.758} C_VEL
LIN {X 0,Y 206.871,Z 468.341,A -85,B 0,C 180,E1 -21165.77,E2 -21165.77} C_VEL
LIN {X 0,Y 206.803,Z 468.349,A -85,B 0,C 180,E1 -21169.867,E2 -21169.867} C_VEL
LIN {X 0,Y 206.766,Z 468.353,A -85,B 0,C 180,E1 -21174.071,E2 -21174.071} C_VEL
LIN {X 0,Y 206.74,Z 468.358,A -85,B 0,C 180,E1 -21178.419,E2 -21178.419} C_VEL
LIN {X 0,Y 206.576,Z 468.38,A -85,B 0,C 180,E1 -21182.979,E2 -21182.979} C_VEL
LIN {X 0,Y 206.299,Z 468.496,A -85,B 0,C 180,E1 -21187.129,E2 -21187.129} C_VEL
LIN {X 0,Y 211.193,Z 483.177,A -85,B 0,C 180,E1 -21188.957,E2 -21188.957} C_VEL
LIN {X 0,Y 214.088,Z 493.813,A -85,B 0,C 180,E1 -21190.416,E2 -21190.416} C_VEL
LIN {X 0,Y 216.771,Z 506.064,A -85,B 0,C 180,E1 -21192.281,E2 -21192.281} C_VEL
LIN {X 0,Y 218.132,Z 513.275,A -85,B 0,C 180,E1 -21193.507,E2 -21193.507} C_VEL
LIN {X 0,Y 216.19,Z 524.421,A -85,B 0,C 180,E1 -21195.318,E2 -21195.318} C_VEL
LIN {X 0,Y 213.802,Z 536.173,A -85,B 0,C 180,E1 -21197.633,E2 -21197.633} C_VEL
LIN {X 0,Y 211.352,Z 548,A -85,B 0,C 180,E1 -21200.497,E2 -21200.497} C_VEL
LIN {X 0,Y 209.18,Z 558.068,A -85,B 0,C 180,E1 -21203.483,E2 -21203.483} C_VEL
LIN {X 0,Y 207.473,Z 566.674,A -85,B 0,C 180,E1 -21206.601,E2 -21206.601} C_VEL
LIN {X 0,Y 206.217,Z 573.939,A -85,B 0,C 180,E1 -21209.821,E2 -21209.821} C_VEL
LIN {X 0,Y 205.176,Z 580.67,A -85,B 0,C 180,E1 -21213.557,E2 -21213.557} C_VEL
LIN {X 0,Y 204.638,Z 585.206,A -85,B 0,C 180,E1 -21216.737,E2 -21216.737} C_VEL
LIN {X 0,Y 204.358,Z 588.643,A -85,B 0,C 180,E1 -21219.884,E2 -21219.884} C_VEL
LIN {X 0,Y 204.545,Z 591.962,A -85,B 0,C 180,E1 -21224.163,E2 -21224.163} C_VEL
LIN {X 0,Y 205.246,Z 593.649,A -85,B 0,C 180,E1 -21228.144,E2 -21228.144} C_VEL
LIN {X 0,Y 206.641,Z 594.031,A -85,B 0,C 180,E1 -21232.181,E2 -21232.181} C_VEL
LIN {X 0,Y 208.804,Z 593.105,A -85,B 0,C 180,E1 -21236.14,E2 -21236.14} C_VEL
LIN {X 0,Y 211.759,Z 590.903,A -85,B 0,C 180,E1 -21240,E2 -21240} C_VEL
LIN {X 0,Y 215.647,Z 587.392,A -85,B 0,C 180,E1 -21243.737,E2 -21243.737} C_VEL
LIN {X 0,Y 220.309,Z 582.513,A -85,B 0,C 180,E1 -21247.331,E2 -21247.331} C_VEL
LIN {X 0,Y 225.938,Z 576.139,A -85,B 0,C 180,E1 -21250.756,E2 -21250.756} C_VEL
LIN {X 0,Y 232.405,Z 568.075,A -85,B 0,C 180,E1 -21254,E2 -21254} C_VEL
LIN {X 0,Y 238.696,Z 559.393,A -85,B 0,C 180,E1 -21256.682,E2 -21256.682} C_VEL
LIN {X 0,Y 245.659,Z 548.738,A -85,B 0,C 180,E1 -21259.253,E2 -21259.253} C_VEL
LIN {X 0,Y 246.486,Z 547.434,A -85,B 0,C 180,E1 -21259.531,E2 -21259.531} C_VEL
LIN {X 0,Y 246.966,Z 545.83,A -85,B 0,C 180,E1 -21260.103,E2 -21260.103} C_VEL
LIN {X 0,Y 247.23,Z 540.723,A -85,B 0,C 180,E1 -21262.647,E2 -21262.647} C_VEL
LIN {X 0,Y 246.932,Z 536.674,A -85,B 0,C 180,E1 -21265.272,E2 -21265.272} C_VEL
LIN {X 0,Y 246.27,Z 534.151,A -85,B 0,C 180,E1 -21267.791,E2 -21267.791} C_VEL
LIN {X 0,Y 245.55,Z 532.257,A -85,B 0,C 180,E1 -21271.01,E2 -21271.01} C_VEL
LIN {X 0,Y 245.2,Z 531.861,A -85,B 0,C 180,E1 -21273.779,E2 -21273.779} C_VEL
LIN {X 0,Y 245.094,Z 532.888,A -85,B 0,C 180,E1 -21277.025,E2 -21277.025} C_VEL
LIN {X 0,Y 245.169,Z 534.636,A -85,B 0,C 180,E1 -21279.289,E2 -21279.289} C_VEL
LIN {X 0,Y 245.245,Z 537.803,A -85,B 0,C 180,E1 -21281.835,E2 -21281.835} C_VEL
LIN {X 0,Y 245.28,Z 540.384,A -85,B 0,C 180,E1 -21283.446,E2 -21283.446} C_VEL
LIN {X 0,Y 245.019,Z 543.585,A -85,B 0,C 180,E1 -21284.97,E2 -21284.97} C_VEL
LIN {X 0,Y 243.955,Z 549.573,A -85,B 0,C 180,E1 -21287.236,E2 -21287.236} C_VEL
LIN {X 0,Y 242.045,Z 557.047,A -85,B 0,C 180,E1 -21289.674,E2 -21289.674} C_VEL
LIN {X 0,Y 239.43,Z 564.64,A -85,B 0,C 180,E1 -21291.946,E2 -21291.946} C_VEL
LIN {X 0,Y 237.492,Z 569.015,A -85,B 0,C 180,E1 -21293.18,E2 -21293.18} C_VEL
LIN {X 0,Y 230.934,Z 578.971,A -85,B 0,C 180,E1 -21295.737,E2 -21295.737} C_VEL
LIN {X 0,Y 225.052,Z 587.374,A -85,B 0,C 180,E1 -21298.462,E2 -21298.462} C_VEL
LIN {X 0,Y 221.286,Z 592.577,A -85,B 0,C 180,E1 -21300.51,E2 -21300.51} C_VEL
LIN {X 0,Y 220.681,Z 593.435,A -85,B 0,C 180,E1 -21300.888,E2 -21300.888} C_VEL
LIN {X 0,Y 218.13,Z 596.254,A -85,B 0,C 180,E1 -21302.076,E2 -21302.076} C_VEL
LIN {X 0,Y 212.432,Z 600.583,A -85,B 0,C 180,E1 -21303.913,E2 -21303.913} C_VEL
LIN {X 0,Y 206.918,Z 604.316,A -85,B 0,C 180,E1 -21305.911,E2 -21305.911} C_VEL
LIN {X 0,Y 204.71,Z 606.248,A -85,B 0,C 180,E1 -21307.331,E2 -21307.331} C_VEL
LIN {X 0,Y 201.124,Z 610.574,A -85,B 0,C 180,E1 -21311.67,E2 -21311.67} C_VEL
LIN {X 0,Y 198.921,Z 613.191,A -85,B 0,C 180,E1 -21315.682,E2 -21315.682} C_VEL
LIN {X 0,Y 197.785,Z 614.62,A -85,B 0,C 180,E1 -21319.766,E2 -21319.766} C_VEL
LIN {X 0,Y 197.478,Z 614.834,A -85,B 0,C 180,E1 -21323.871,E2 -21323.871} C_VEL
LIN {X 0,Y 197.648,Z 614.473,A -85,B 0,C 180,E1 -21325.922,E2 -21325.922} C_VEL
LIN {X 0,Y 197.894,Z 612.72,A -85,B 0,C 180,E1 -21330,E2 -21330} C_VEL
LIN {X 0,Y 197.822,Z 609.464,A -85,B 0,C 180,E1 -21334.074,E2 -21334.074} C_VEL
LIN {X 0,Y 197.898,Z 605.971,A -85,B 0,C 180,E1 -21337.14,E2 -21337.14} C_VEL
LIN {X 0,Y 198.125,Z 601.483,A -85,B 0,C 180,E1 -21340.216,E2 -21340.216} C_VEL
LIN {X 0,Y 198.912,Z 594.916,A -85,B 0,C 180,E1 -21343.797,E2 -21343.797} C_VEL
LIN {X 0,Y 200.207,Z 586.677,A -85,B 0,C 180,E1 -21347.36,E2 -21347.36} C_VEL
LIN {X 0,Y 201.943,Z 578.147,A -85,B 0,C 180,E1 -21350.366,E2 -21350.366} C_VEL
LIN {X 0,Y 204.119,Z 567.892,A -85,B 0,C 180,E1 -21353.325,E2 -21353.325} C_VEL
LIN {X 0,Y 206.663,Z 556.649,A -85,B 0,C 180,E1 -21355.966,E2 -21355.966} C_VEL
LIN {X 0,Y 207.946,Z 550.781,A -85,B 0,C 180,E1 -21357.146,E2 -21357.146} C_VEL
LIN {X 0,Y 207.493,Z 541.857,A -85,B 0,C 180,E1 -21358.858,E2 -21358.858} C_VEL
LIN {X 0,Y 206.416,Z 528.514,A -85,B 0,C 180,E1 -21361.083,E2 -21361.083} C_VEL
LIN {X 0,Y 205.083,Z 515.633,A -85,B 0,C 180,E1 -21362.905,E2 -21362.905} C_VEL
LIN {X 0,Y 203.09,Z 500.267,A -85,B 0,C 180,E1 -21364.728,E2 -21364.728} C_VEL
LIN {X 0,Y 201.029,Z 486.165,A -85,B 0,C 180,E1 -21366.092,E2 -21366.092} C_VEL
LIN {X 0,Y 201.843,Z 482.414,A -85,B 0,C 180,E1 -21370.003,E2 -21370.003} C_VEL
LIN {X 0,Y 201.685,Z 479.675,A -85,B 0,C 180,E1 -21372.965,E2 -21372.965} C_VEL
LIN {X 0,Y 200.971,Z 475.904,A -85,B 0,C 180,E1 -21377.253,E2 -21377.253} C_VEL
LIN {X 0,Y 200.193,Z 471.844,A -85,B 0,C 180,E1 -21382.095,E2 -21382.095} C_VEL
LIN {X 0,Y 199.773,Z 469.223,A -85,B 0,C 180,E1 -21385.446,E2 -21385.446} C_VEL
LIN {X 0,Y 199.673,Z 469.239,A -85,B 0,C 180,E1 -21390.478,E2 -21390.478} C_VEL
LIN {X 0,Y 199.67,Z 469.233,A -85,B 0,C 180,E1 -21395.016,E2 -21395.016} C_VEL
LIN {X 0,Y 199.706,Z 469.233,A -85,B 0,C 180,E1 -21399.396,E2 -21399.396} C_VEL
LIN {X 0,Y 199.835,Z 469.215,A -85,B 0,C 180,E1 -21401.722,E2 -21401.722} C_VEL
LIN {X 0,Y 199.845,Z 469.213,A -85,B 0,C 180,E1 -21405.749,E2 -21405.749} C_VEL
LIN {X 0,Y 200.068,Z 469.187,A -85,B 0,C 180,E1 -21409.884,E2 -21409.884} C_VEL
LIN {X 0,Y 200.032,Z 469.188,A -85,B 0,C 180,E1 -21413.95,E2 -21413.95} C_VEL
LIN {X 0,Y 200.319,Z 469.156,A -85,B 0,C 180,E1 -21417.99,E2 -21417.99} C_VEL
LIN {X 0,Y 200.476,Z 469.136,A -85,B 0,C 180,E1 -21420,E2 -21420} C_VEL
LIN {X 0,Y 200.033,Z 469.19,A -85,B 0,C 180,E1 -21424.03,E2 -21424.03} C_VEL
LIN {X 0,Y 200.109,Z 469.183,A -85,B 0,C 180,E1 -21428.076,E2 -21428.076} C_VEL
LIN {X 0,Y 199.911,Z 469.205,A -85,B 0,C 180,E1 -21432.178,E2 -21432.178} C_VEL
LIN {X 0,Y 199.802,Z 469.223,A -85,B 0,C 180,E1 -21436.344,E2 -21436.344} C_VEL
LIN {X 0,Y 199.698,Z 469.233,A -85,B 0,C 180,E1 -21440.606,E2 -21440.606} C_VEL
LIN {X 0,Y 199.672,Z 469.236,A -85,B 0,C 180,E1 -21444.985,E2 -21444.985} C_VEL
LIN {X 0,Y 199.674,Z 469.233,A -85,B 0,C 180,E1 -21449.523,E2 -21449.523} C_VEL
LIN {X 0,Y 199.663,Z 469.24,A -85,B 0,C 180,E1 -21452.353,E2 -21452.353} C_VEL
LIN {X 0,Y 199.639,Z 469.236,A -85,B 0,C 180,E1 -21456.76,E2 -21456.76} C_VEL
LIN {X 0,Y 199.638,Z 469.239,A -85,B 0,C 180,E1 -21459.322,E2 -21459.322} C_VEL
LIN {X 0,Y 199.594,Z 469.243,A -85,B 0,C 180,E1 -21464.768,E2 -21464.768} C_VEL
LIN {X 0,Y 199.608,Z 469.246,A -85,B 0,C 180,E1 -21468.013,E2 -21468.013} C_VEL
LIN {X 0,Y 199.643,Z 469.24,A -85,B 0,C 180,E1 -21470.757,E2 -21470.757} C_VEL
LIN {X 0,Y 199.636,Z 469.239,A -85,B 0,C 180,E1 -21475.719,E2 -21475.719} C_VEL
LIN {X 0,Y 199.706,Z 469.234,A -85,B 0,C 180,E1 -21478.139,E2 -21478.139} C_VEL
LIN {X 0,Y 199.689,Z 469.231,A -85,B 0,C 180,E1 -21482.773,E2 -21482.773} C_VEL
LIN {X 0,Y 199.741,Z 469.229,A -85,B 0,C 180,E1 -21487.23,E2 -21487.23} C_VEL
LIN {X 0,Y 199.799,Z 469.219,A -85,B 0,C 180,E1 -21491.758,E2 -21491.758} C_VEL
LIN {X 0,Y 199.839,Z 469.218,A -85,B 0,C 180,E1 -21495.749,E2 -21495.749} C_VEL
LIN {X 0,Y 200.025,Z 469.19,A -85,B 0,C 180,E1 -21499.882,E2 -21499.882} C_VEL
LIN {X 0,Y 200.018,Z 469.194,A -85,B 0,C 180,E1 -21503.949,E2 -21503.949} C_VEL
LIN {X 0,Y 200.323,Z 469.154,A -85,B 0,C 180,E1 -21507.989,E2 -21507.989} C_VEL
LIN {X 0,Y 200.483,Z 469.132,A -85,B 0,C 180,E1 -21510,E2 -21510} C_VEL
LIN {X 0,Y 200.033,Z 469.192,A -85,B 0,C 180,E1 -21514.029,E2 -21514.029} C_VEL
LIN {X 0,Y 200.099,Z 469.179,A -85,B 0,C 180,E1 -21518.076,E2 -21518.076} C_VEL
LIN {X 0,Y 199.882,Z 469.21,A -85,B 0,C 180,E1 -21522.179,E2 -21522.179} C_VEL
LIN {X 0,Y 199.809,Z 469.22,A -85,B 0,C 180,E1 -21526.343,E2 -21526.343} C_VEL
LIN {X 0,Y 199.827,Z 469.216,A -85,B 0,C 180,E1 -21528.453,E2 -21528.453} C_VEL
LIN {X 0,Y 199.739,Z 469.228,A -85,B 0,C 180,E1 -21533.817,E2 -21533.817} C_VEL
LIN {X 0,Y 199.711,Z 469.234,A -85,B 0,C 180,E1 -21538.384,E2 -21538.384} C_VEL
LIN {X 0,Y 199.562,Z 469.252,A -85,B 0,C 180,E1 -21542.304,E2 -21542.304} C_VEL
LIN {X 0,Y 199.304,Z 469.284,A -85,B 0,C 180,E1 -21546.346,E2 -21546.346} C_VEL
LIN {X 0,Y 205.038,Z 486.692,A -85,B 0,C 180,E1 -21548.699,E2 -21548.699} C_VEL
LIN {X 0,Y 208.082,Z 498.633,A -85,B 0,C 180,E1 -21550.474,E2 -21550.474} C_VEL
LIN {X 0,Y 210.632,Z 511.206,A -85,B 0,C 180,E1 -21552.56,E2 -21552.56} C_VEL
LIN {X 0,Y 211.127,Z 515.086,A -85,B 0,C 180,E1 -21553.249,E2 -21553.249} C_VEL
LIN {X 0,Y 208.501,Z 528.649,A -85,B 0,C 180,E1 -21555.618,E2 -21555.618} C_VEL
LIN {X 0,Y 206.1,Z 540.083,A -85,B 0,C 180,E1 -21558.083,E2 -21558.083} C_VEL
LIN {X 0,Y 203.738,Z 551.044,A -85,B 0,C 180,E1 -21560.983,E2 -21560.983} C_VEL
LIN {X 0,Y 201.502,Z 561.122,A -85,B 0,C 180,E1 -21564.252,E2 -21564.252} C_VEL
LIN {X 0,Y 199.929,Z 569.354,A -85,B 0,C 180,E1 -21567.527,E2 -21567.527} C_VEL
LIN {X 0,Y 198.755,Z 576.255,A -85,B 0,C 180,E1 -21570.9,E2 -21570.9} C_VEL
LIN {X 0,Y 197.842,Z 582.56,A -85,B 0,C 180,E1 -21574.768,E2 -21574.768} C_VEL
LIN {X 0,Y 197.418,Z 586.407,A -85,B 0,C 180,E1 -21577.754,E2 -21577.754} C_VEL
LIN {X 0,Y 197.244,Z 589.954,A -85,B 0,C 180,E1 -21581.296,E2 -21581.296} C_VEL
LIN {X 0,Y 197.613,Z 592.842,A -85,B 0,C 180,E1 -21585.584,E2 -21585.584} C_VEL
LIN {X 0,Y 198.622,Z 594.31,A -85,B 0,C 180,E1 -21589.809,E2 -21589.809} C_VEL
LIN {X 0,Y 200.34,Z 594.453,A -85,B 0,C 180,E1 -21593.959,E2 -21593.959} C_VEL
LIN {X 0,Y 202.976,Z 593.305,A -85,B 0,C 180,E1 -21598.015,E2 -21598.015} C_VEL
LIN {X 0,Y 206.39,Z 590.904,A -85,B 0,C 180,E1 -21601.951,E2 -21601.951} C_VEL
LIN {X 0,Y 210.786,Z 587.192,A -85,B 0,C 180,E1 -21605.74,E2 -21605.74} C_VEL
LIN {X 0,Y 216.031,Z 582.117,A -85,B 0,C 180,E1 -21609.361,E2 -21609.361} C_VEL
LIN {X 0,Y 222.218,Z 575.508,A -85,B 0,C 180,E1 -21612.79,E2 -21612.79} C_VEL
LIN {X 0,Y 228.366,Z 568.289,A -85,B 0,C 180,E1 -21615.621,E2 -21615.621} C_VEL
LIN {X 0,Y 235.986,Z 558.282,A -85,B 0,C 180,E1 -21618.672,E2 -21618.672} C_VEL
LIN {X 0,Y 241.232,Z 550.757,A -85,B 0,C 180,E1 -21620.463,E2 -21620.463} C_VEL
LIN {X 0,Y 241.761,Z 549.556,A -85,B 0,C 180,E1 -21620.862,E2 -21620.862} C_VEL
LIN {X 0,Y 242.3,Z 544.989,A -85,B 0,C 180,E1 -21623.372,E2 -21623.372} C_VEL
LIN {X 0,Y 242.235,Z 541.495,A -85,B 0,C 180,E1 -21625.922,E2 -21625.922} C_VEL
LIN {X 0,Y 241.923,Z 539.858,A -85,B 0,C 180,E1 -21627.698,E2 -21627.698} C_VEL
LIN {X 0,Y 241.518,Z 538.584,A -85,B 0,C 180,E1 -21629.649,E2 -21629.649} C_VEL
LIN {X 0,Y 241.168,Z 537.682,A -85,B 0,C 180,E1 -21632.319,E2 -21632.319} C_VEL
LIN {X 0,Y 240.932,Z 537.931,A -85,B 0,C 180,E1 -21635.239,E2 -21635.239} C_VEL
LIN {X 0,Y 240.858,Z 539.399,A -85,B 0,C 180,E1 -21638.018,E2 -21638.018} C_VEL
LIN {X 0,Y 240.773,Z 542.755,A -85,B 0,C 180,E1 -21641.179,E2 -21641.179} C_VEL
LIN {X 0,Y 240.654,Z 545.674,A -85,B 0,C 180,E1 -21643.107,E2 -21643.107} C_VEL
LIN {X 0,Y 240.127,Z 548.797,A -85,B 0,C 180,E1 -21644.622,E2 -21644.622} C_VEL
LIN {X 0,Y 238.296,Z 555.727,A -85,B 0,C 180,E1 -21647.287,E2 -21647.287} C_VEL
LIN {X 0,Y 235.891,Z 562.645,A -85,B 0,C 180,E1 -21649.609,E2 -21649.609} C_VEL
LIN {X 0,Y 232.687,Z 569.829,A -85,B 0,C 180,E1 -21651.837,E2 -21651.837} C_VEL
LIN {X 0,Y 228.056,Z 576.582,A -85,B 0,C 180,E1 -21653.614,E2 -21653.614} C_VEL
LIN {X 0,Y 221.642,Z 585.253,A -85,B 0,C 180,E1 -21656.297,E2 -21656.297} C_VEL
LIN {X 0,Y 216.608,Z 591.566,A -85,B 0,C 180,E1 -21658.727,E2 -21658.727} C_VEL
LIN {X 0,Y 211.035,Z 598.668,A -85,B 0,C 180,E1 -21662.21,E2 -21662.21} C_VEL
LIN {X 0,Y 206.277,Z 604.374,A -85,B 0,C 180,E1 -21665.868,E2 -21665.868} C_VEL
LIN {X 0,Y 204.71,Z 606.248,A -85,B 0,C 180,E1 -21667.331,E2 -21667.331} C_VEL
LIN {X 0,Y 202.642,Z 608.019,A -85,B 0,C 180,E1 -21668.811,E2 -21668.811} C_VEL
LIN {X 0,Y 197.828,Z 610.462,A -85,B 0,C 180,E1 -21671.192,E2 -21671.192} C_VEL
LIN {X 0,Y 193.371,Z 612.309,A -85,B 0,C 180,E1 -21673.725,E2 -21673.725} C_VEL
LIN {X 0,Y 191.91,Z 613.083,A -85,B 0,C 180,E1 -21675.409,E2 -21675.409} C_VEL
LIN {X 0,Y 190.754,Z 614.219,A -85,B 0,C 180,E1 -21679.385,E2 -21679.385} C_VEL
LIN {X 0,Y 190.414,Z 614.245,A -85,B 0,C 180,E1 -21683.643,E2 -21683.643} C_VEL
LIN {X 0,Y 190.581,Z 613.806,A -85,B 0,C 180,E1 -21685.77,E2 -21685.77} C_VEL
LIN {X 0,Y 190.848,Z 611.884,A -85,B 0,C 180,E1 -21690,E2 -21690} C_VEL
LIN {X 0,Y 190.78,Z 608.441,A -85,B 0,C 180,E1 -21694.225,E2 -21694.225} C_VEL
LIN {X 0,Y 190.863,Z 604.767,A -85,B 0,C 180,E1 -21697.405,E2 -21697.405} C_VEL
LIN {X 0,Y 191.332,Z 598.369,A -85,B 0,C 180,E1 -21701.655,E2 -21701.655} C_VEL
LIN {X 0,Y 192.274,Z 591.154,A -85,B 0,C 180,E1 -21705.367,E2 -21705.367} C_VEL
LIN {X 0,Y 193.958,Z 582.158,A -85,B 0,C 180,E1 -21709.033,E2 -21709.033} C_VEL
LIN {X 0,Y 195.988,Z 572.822,A -85,B 0,C 180,E1 -21712.118,E2 -21712.118} C_VEL
LIN {X 0,Y 198.542,Z 561.59,A -85,B 0,C 180,E1 -21715.136,E2 -21715.136} C_VEL
LIN {X 0,Y 200.959,Z 550.515,A -85,B 0,C 180,E1 -21717.559,E2 -21717.559} C_VEL
LIN {X 0,Y 200.223,Z 537.993,A -85,B 0,C 180,E1 -21720.012,E2 -21720.012} C_VEL
LIN {X 0,Y 199.093,Z 524.646,A -85,B 0,C 180,E1 -21722.233,E2 -21722.233} C_VEL
LIN {X 0,Y 197.469,Z 509.947,A -85,B 0,C 180,E1 -21724.28,E2 -21724.28} C_VEL
LIN {X 0,Y 195.349,Z 494.26,A -85,B 0,C 180,E1 -21726.074,E2 -21726.074} C_VEL
LIN {X 0,Y 194.123,Z 485.753,A -85,B 0,C 180,E1 -21726.926,E2 -21726.926} C_VEL
LIN {X 0,Y 194.765,Z 482.456,A -85,B 0,C 180,E1 -21730.505,E2 -21730.505} C_VEL
LIN {X 0,Y 194.486,Z 479.636,A -85,B 0,C 180,E1 -21733.72,E2 -21733.72} C_VEL
LIN {X 0,Y 193.813,Z 476.121,A -85,B 0,C 180,E1 -21737.868,E2 -21737.868} C_VEL
LIN {X 0,Y 192.983,Z 471.843,A -85,B 0,C 180,E1 -21743.243,E2 -21743.243} C_VEL
LIN {X 0,Y 192.732,Z 470.099,A -85,B 0,C 180,E1 -21745.584,E2 -21745.584} C_VEL
LIN {X 0,Y 192.662,Z 470.109,A -85,B 0,C 180,E1 -21751.692,E2 -21751.692} C_VEL
LIN {X 0,Y 192.703,Z 470.101,A -85,B 0,C 180,E1 -21756.349,E2 -21756.349} C_VEL
LIN {X 0,Y 192.779,Z 470.095,A -85,B 0,C 180,E1 -21761.414,E2 -21761.414} C_VEL
LIN {X 0,Y 192.85,Z 470.087,A -85,B 0,C 180,E1 -21767.37,E2 -21767.37} C_VEL
LIN {X 0,Y 193.059,Z 470.058,A -85,B 0,C 180,E1 -21771.628,E2 -21771.628} C_VEL
LIN {X 0,Y 193.261,Z 470.035,A -85,B 0,C 180,E1 -21777.916,E2 -21777.916} C_VEL
LIN {X 0,Y 193.44,Z 470.012,A -85,B 0,C 180,E1 -21780,E2 -21780} C_VEL
LIN {X 0,Y 192.979,Z 470.07,A -85,B 0,C 180,E1 -21784.177,E2 -21784.177} C_VEL
LIN {X 0,Y 193.06,Z 470.062,A -85,B 0,C 180,E1 -21788.373,E2 -21788.373} C_VEL
LIN {X 0,Y 192.85,Z 470.088,A -85,B 0,C 180,E1 -21792.631,E2 -21792.631} C_VEL
LIN {X 0,Y 192.755,Z 470.097,A -85,B 0,C 180,E1 -21796.959,E2 -21796.959} C_VEL
LIN {X 0,Y 192.634,Z 470.111,A -85,B 0,C 180,E1 -21801.398,E2 -21801.398} C_VEL
LIN {X 0,Y 192.663,Z 470.113,A -85,B 0,C 180,E1 -21804.225,E2 -21804.225} C_VEL
LIN {X 0,Y 192.649,Z 470.108,A -85,B 0,C 180,E1 -21808.893,E2 -21808.893} C_VEL
LIN {X 0,Y 192.599,Z 470.117,A -85,B 0,C 180,E1 -21813.186,E2 -21813.186} C_VEL
LIN {X 0,Y 192.608,Z 470.112,A -85,B 0,C 180,E1 -21816.608,E2 -21816.608} C_VEL
LIN {X 0,Y 192.522,Z 470.127,A -85,B 0,C 180,E1 -21821.079,E2 -21821.079} C_VEL
LIN {X 0,Y 192.533,Z 470.124,A -85,B 0,C 180,E1 -21826.089,E2 -21826.089} C_VEL
LIN {X 0,Y 192.55,Z 470.126,A -85,B 0,C 180,E1 -21830.041,E2 -21830.041} C_VEL
LIN {X 0,Y 192.599,Z 470.114,A -85,B 0,C 180,E1 -21834.279,E2 -21834.279} C_VEL
LIN {X 0,Y 192.61,Z 470.117,A -85,B 0,C 180,E1 -21839.281,E2 -21839.281} C_VEL
LIN {X 0,Y 192.667,Z 470.11,A -85,B 0,C 180,E1 -21841.693,E2 -21841.693} C_VEL
LIN {X 0,Y 192.708,Z 470.104,A -85,B 0,C 180,E1 -21846.349,E2 -21846.349} C_VEL
LIN {X 0,Y 192.735,Z 470.1,A -85,B 0,C 180,E1 -21851.458,E2 -21851.458} C_VEL
LIN {X 0,Y 192.767,Z 470.097,A -85,B 0,C 180,E1 -21855.214,E2 -21855.214} C_VEL
LIN {X 0,Y 192.948,Z 470.073,A -85,B 0,C 180,E1 -21859.567,E2 -21859.567} C_VEL
LIN {X 0,Y 192.98,Z 470.072,A -85,B 0,C 180,E1 -21863.728,E2 -21863.728} C_VEL
LIN {X 0,Y 193.265,Z 470.033,A -85,B 0,C 180,E1 -21867.916,E2 -21867.916} C_VEL
LIN {X 0,Y 193.447,Z 470.008,A -85,B 0,C 180,E1 -21870,E2 -21870} C_VEL
LIN {X 0,Y 192.979,Z 470.07,A -85,B 0,C 180,E1 -21874.177,E2 -21874.177} C_VEL
LIN {X 0,Y 193.045,Z 470.058,A -85,B 0,C 180,E1 -21878.373,E2 -21878.373} C_VEL
LIN {X 0,Y 192.808,Z 470.092,A -85,B 0,C 180,E1 -21882.633,E2 -21882.633} C_VEL
LIN {X 0,Y 192.774,Z 470.097,A -85,B 0,C 180,E1 -21886.957,E2 -21886.957} C_VEL
LIN {X 0,Y 192.645,Z 470.113,A -85,B 0,C 180,E1 -21891.396,E2 -21891.396} C_VEL
LIN {X 0,Y 192.667,Z 470.109,A -85,B 0,C 180,E1 -21894.224,E2 -21894.224} C_VEL
LIN {X 0,Y 192.642,Z 470.116,A -85,B 0,C 180,E1 -21898.886,E2 -21898.886} C_VEL
LIN {X 0,Y 192.399,Z 470.144,A -85,B 0,C 180,E1 -21904.484,E2 -21904.484} C_VEL
LIN {X 0,Y 192.317,Z 470.154,A -85,B 0,C 180,E1 -21905.62,E2 -21905.62} C_VEL
LIN {X 0,Y 198.075,Z 487.62,A -85,B 0,C 180,E1 -21908.06,E2 -21908.06} C_VEL
LIN {X 0,Y 200.777,Z 497.805,A -85,B 0,C 180,E1 -21909.637,E2 -21909.637} C_VEL
LIN {X 0,Y 203.306,Z 509.97,A -85,B 0,C 180,E1 -21911.716,E2 -21911.716} C_VEL
LIN {X 0,Y 204.214,Z 515.041,A -85,B 0,C 180,E1 -21912.657,E2 -21912.657} C_VEL
LIN {X 0,Y 202.223,Z 525.884,A -85,B 0,C 180,E1 -21914.565,E2 -21914.565} C_VEL
LIN {X 0,Y 199.49,Z 538.659,A -85,B 0,C 180,E1 -21917.298,E2 -21917.298} C_VEL
LIN {X 0,Y 196.943,Z 550.362,A -85,B 0,C 180,E1 -21920.399,E2 -21920.399} C_VEL
LIN {X 0,Y 194.777,Z 559.737,A -85,B 0,C 180,E1 -21923.461,E2 -21923.461} C_VEL
LIN {X 0,Y 193.055,Z 568.356,A -85,B 0,C 180,E1 -21926.902,E2 -21926.902} C_VEL
LIN {X 0,Y 191.827,Z 575.437,A -85,B 0,C 180,E1 -21930.356,E2 -21930.356} C_VEL
LIN {X 0,Y 190.933,Z 581.186,A -85,B 0,C 180,E1 -21933.787,E2 -21933.787} C_VEL
LIN {X 0,Y 190.382,Z 585.948,A -85,B 0,C 180,E1 -21937.348,E2 -21937.348} C_VEL
LIN {X 0,Y 190.135,Z 589.288,A -85,B 0,C 180,E1 -21940.569,E2 -21940.569} C_VEL
LIN {X 0,Y 190.431,Z 592.624,A -85,B 0,C 180,E1 -21945.028,E2 -21945.028} C_VEL
LIN {X 0,Y 191.383,Z 594.531,A -85,B 0,C 180,E1 -21949.419,E2 -21949.419} C_VEL
LIN {X 0,Y 193.107,Z 595.094,A -85,B 0,C 180,E1 -21953.731,E2 -21953.731} C_VEL
LIN {X 0,Y 195.726,Z 594.372,A -85,B 0,C 180,E1 -21957.942,E2 -21957.942} C_VEL
LIN {X 0,Y 199.185,Z 592.401,A -85,B 0,C 180,E1 -21962.022,E2 -21962.022} C_VEL
LIN {X 0,Y 203.685,Z 589.149,A -85,B 0,C 180,E1 -21965.941,E2 -21965.941} C_VEL
LIN {X 0,Y 209.008,Z 584.559,A -85,B 0,C 180,E1 -21969.679,E2 -21969.679} C_VEL
LIN {X 0,Y 215.359,Z 578.5,A -85,B 0,C 180,E1 -21973.205,E2 -21973.205} C_VEL
LIN {X 0,Y 222.571,Z 570.828,A -85,B 0,C 180,E1 -21976.51,E2 -21976.51} C_VEL
LIN {X 0,Y 229.481,Z 562.638,A -85,B 0,C 180,E1 -21979.221,E2 -21979.221} C_VEL
LIN {X 0,Y 236.604,Z 553.286,A -85,B 0,C 180,E1 -21981.654,E2 -21981.654} C_VEL
LIN {X 0,Y 237.139,Z 550.496,A -85,B 0,C 180,E1 -21983.26,E2 -21983.26} C_VEL
LIN {X 0,Y 237.45,Z 547.395,A -85,B 0,C 180,E1 -21985.512,E2 -21985.512} C_VEL
LIN {X 0,Y 237.249,Z 544.929,A -85,B 0,C 180,E1 -21988.292,E2 -21988.292} C_VEL
LIN {X 0,Y 236.915,Z 543.748,A -85,B 0,C 180,E1 -21990.655,E2 -21990.655} C_VEL
LIN {X 0,Y 236.804,Z 543.263,A -85,B 0,C 180,E1 -21992.29,E2 -21992.29} C_VEL
LIN {X 0,Y 236.644,Z 543.385,A -85,B 0,C 180,E1 -21994.352,E2 -21994.352} C_VEL
LIN {X 0,Y 236.486,Z 544.253,A -85,B 0,C 180,E1 -21996.642,E2 -21996.642} C_VEL
LIN {X 0,Y 236.27,Z 546.368,A -85,B 0,C 180,E1 -21999.342,E2 -21999.342} C_VEL
LIN {X 0,Y 236.078,Z 549.409,A -85,B 0,C 180,E1 -22001.907,E2 -22001.907} C_VEL
LIN {X 0,Y 235.61,Z 551.807,A -85,B 0,C 180,E1 -22003.319,E2 -22003.319} C_VEL
LIN {X 0,Y 234.167,Z 556.58,A -85,B 0,C 180,E1 -22005.389,E2 -22005.389} C_VEL
LIN {X 0,Y 231.957,Z 562.463,A -85,B 0,C 180,E1 -22007.619,E2 -22007.619} C_VEL
LIN {X 0,Y 228.907,Z 568.982,A -85,B 0,C 180,E1 -22009.854,E2 -22009.854} C_VEL
LIN {X 0,Y 226.723,Z 572.828,A -85,B 0,C 180,E1 -22011.059,E2 -22011.059} C_VEL
LIN {X 0,Y 219.588,Z 582.003,A -85,B 0,C 180,E1 -22013.695,E2 -22013.695} C_VEL
LIN {X 0,Y 213.997,Z 588.658,A -85,B 0,C 180,E1 -22016.062,E2 -22016.062} C_VEL
LIN {X 0,Y 209.149,Z 594.384,A -85,B 0,C 180,E1 -22018.612,E2 -22018.612} C_VEL
LIN {X 0,Y 203.446,Z 600.79,A -85,B 0,C 180,E1 -22022.203,E2 -22022.203} C_VEL
LIN {X 0,Y 198.728,Z 605.907,A -85,B 0,C 180,E1 -22026.003,E2 -22026.003} C_VEL
LIN {X 0,Y 195.896,Z 608.95,A -85,B 0,C 180,E1 -22028.976,E2 -22028.976} C_VEL
LIN {X 0,Y 193.083,Z 611.943,A -85,B 0,C 180,E1 -22033.071,E2 -22033.071} C_VEL
LIN {X 0,Y 191.91,Z 613.083,A -85,B 0,C 180,E1 -22035.409,E2 -22035.409} C_VEL
LIN {X 0,Y 190.617,Z 613.693,A -85,B 0,C 180,E1 -22037.13,E2 -22037.13} C_VEL
LIN {X 0,Y 187.095,Z 614.068,A -85,B 0,C 180,E1 -22039.942,E2 -22039.942} C_VEL
LIN {X 0,Y 184.46,Z 613.857,A -85,B 0,C 180,E1 -22042.259,E2 -22042.259} C_VEL
LIN {X 0,Y 183.437,Z 613.493,A -85,B 0,C 180,E1 -22044.076,E2 -22044.076} C_VEL
LIN {X 0,Y 183.394,Z 613.331,A -85,B 0,C 180,E1 -22044.692,E2 -22044.692} C_VEL
LIN {X 0,Y 183.553,Z 612.226,A -85,B 0,C 180,E1 -22047.806,E2 -22047.806} C_VEL
LIN {X 0,Y 183.802,Z 611.022,A -85,B 0,C 180,E1 -22050,E2 -22050} C_VEL
LIN {X 0,Y 183.744,Z 607.366,A -85,B 0,C 180,E1 -22054.387,E2 -22054.387} C_VEL
LIN {X 0,Y 183.823,Z 603.543,A -85,B 0,C 180,E1 -22057.69,E2 -22057.69} C_VEL
LIN {X 0,Y 184.133,Z 598.698,A -85,B 0,C 180,E1 -22061.002,E2 -22061.002} C_VEL
LIN {X 0,Y 185.064,Z 591.706,A -85,B 0,C 180,E1 -22064.853,E2 -22064.853} C_VEL
LIN {X 0,Y 186.624,Z 583.042,A -85,B 0,C 180,E1 -22068.669,E2 -22068.669} C_VEL
LIN {X 0,Y 188.617,Z 574.042,A -85,B 0,C 180,E1 -22071.876,E2 -22071.876} C_VEL
LIN {X 0,Y 191.071,Z 563.166,A -85,B 0,C 180,E1 -22075.023,E2 -22075.023} C_VEL
LIN {X 0,Y 193.588,Z 552.299,A -85,B 0,C 180,E1 -22077.572,E2 -22077.572} C_VEL
LIN {X 0,Y 193.924,Z 549.792,A -85,B 0,C 180,E1 -22078.107,E2 -22078.107} C_VEL
LIN {X 0,Y 193.168,Z 537.429,A -85,B 0,C 180,E1 -22080.621,E2 -22080.621} C_VEL
LIN {X 0,Y 192.19,Z 525.107,A -85,B 0,C 180,E1 -22082.748,E2 -22082.748} C_VEL
LIN {X 0,Y 190.707,Z 511.298,A -85,B 0,C 180,E1 -22084.772,E2 -22084.772} C_VEL
LIN {X 0,Y 188.725,Z 495.949,A -85,B 0,C 180,E1 -22086.625,E2 -22086.625} C_VEL
LIN {X 0,Y 187.221,Z 485.44,A -85,B 0,C 180,E1 -22087.703,E2 -22087.703} C_VEL
LIN {X 0,Y 187.568,Z 483.788,A -85,B 0,C 180,E1 -22089.566,E2 -22089.566} C_VEL
LIN {X 0,Y 187.598,Z 481.327,A -85,B 0,C 180,E1 -22092.401,E2 -22092.401} C_VEL
LIN {X 0,Y 186.832,Z 477.249,A -85,B 0,C 180,E1 -22097.383,E2 -22097.383} C_VEL
LIN {X 0,Y 185.994,Z 473.037,A -85,B 0,C 180,E1 -22102.802,E2 -22102.802} C_VEL
LIN {X 0,Y 185.673,Z 470.978,A -85,B 0,C 180,E1 -22105.707,E2 -22105.707} C_VEL
LIN {X 0,Y 185.58,Z 470.995,A -85,B 0,C 180,E1 -22110.576,E2 -22110.576} C_VEL
LIN {X 0,Y 185.585,Z 470.988,A -85,B 0,C 180,E1 -22115.383,E2 -22115.383} C_VEL
LIN {X 0,Y 185.692,Z 470.979,A -85,B 0,C 180,E1 -22121.116,E2 -22121.116} C_VEL
LIN {X 0,Y 185.725,Z 470.971,A -85,B 0,C 180,E1 -22124.64,E2 -22124.64} C_VEL
LIN {X 0,Y 185.922,Z 470.949,A -85,B 0,C 180,E1 -22129.359,E2 -22129.359} C_VEL
LIN {X 0,Y 185.959,Z 470.941,A -85,B 0,C 180,E1 -22133.49,E2 -22133.49} C_VEL
LIN {X 0,Y 186.206,Z 470.914,A -85,B 0,C 180,E1 -22137.837,E2 -22137.837} C_VEL
LIN {X 0,Y 186.404,Z 470.888,A -85,B 0,C 180,E1 -22140,E2 -22140} C_VEL
LIN {X 0,Y 185.926,Z 470.949,A -85,B 0,C 180,E1 -22144.336,E2 -22144.336} C_VEL
LIN {X 0,Y 186.007,Z 470.938,A -85,B 0,C 180,E1 -22148.693,E2 -22148.693} C_VEL
LIN {X 0,Y 185.761,Z 470.969,A -85,B 0,C 180,E1 -22153.121,E2 -22153.121} C_VEL
LIN {X 0,Y 185.673,Z 470.976,A -85,B 0,C 180,E1 -22158.867,E2 -22158.867} C_VEL
LIN {X 0,Y 185.6,Z 470.99,A -85,B 0,C 180,E1 -22164.663,E2 -22164.663} C_VEL
LIN {X 0,Y 185.578,Z 470.989,A -85,B 0,C 180,E1 -22169.494,E2 -22169.494} C_VEL
LIN {X 0,Y 185.518,Z 470.999,A -85,B 0,C 180,E1 -22174.629,E2 -22174.629} C_VEL
LIN {X 0,Y 185.543,Z 470.991,A -85,B 0,C 180,E1 -22177.305,E2 -22177.305} C_VEL
LIN {X 0,Y 185.484,Z 471.004,A -85,B 0,C 180,E1 -22180.73,E2 -22180.73} C_VEL
LIN {X 0,Y 185.499,Z 471,A -85,B 0,C 180,E1 -22186.043,E2 -22186.043} C_VEL
LIN {X 0,Y 185.5,Z 471.005,A -85,B 0,C 180,E1 -22189.904,E2 -22189.904} C_VEL
LIN {X 0,Y 185.545,Z 470.994,A -85,B 0,C 180,E1 -22192.697,E2 -22192.697} C_VEL
LIN {X 0,Y 185.547,Z 470.998,A -85,B 0,C 180,E1 -22197.976,E2 -22197.976} C_VEL
LIN {X 0,Y 185.584,Z 470.991,A -85,B 0,C 180,E1 -22200.577,E2 -22200.577} C_VEL
LIN {X 0,Y 185.59,Z 470.989,A -85,B 0,C 180,E1 -22205.383,E2 -22205.383} C_VEL
LIN {X 0,Y 185.678,Z 470.978,A -85,B 0,C 180,E1 -22211.133,E2 -22211.133} C_VEL
LIN {X 0,Y 185.698,Z 470.976,A -85,B 0,C 180,E1 -22214.638,E2 -22214.638} C_VEL
LIN {X 0,Y 185.891,Z 470.953,A -85,B 0,C 180,E1 -22219.419,E2 -22219.419} C_VEL
LIN {X 0,Y 185.943,Z 470.948,A -85,B 0,C 180,E1 -22223.489,E2 -22223.489} C_VEL
LIN {X 0,Y 186.208,Z 470.912,A -85,B 0,C 180,E1 -22227.837,E2 -22227.837} C_VEL
LIN {X 0,Y 186.41,Z 470.885,A -85,B 0,C 180,E1 -22230,E2 -22230} C_VEL
LIN {X 0,Y 185.926,Z 470.949,A -85,B 0,C 180,E1 -22234.336,E2 -22234.336} C_VEL
LIN {X 0,Y 185.99,Z 470.937,A -85,B 0,C 180,E1 -22238.693,E2 -22238.693} C_VEL
LIN {X 0,Y 185.734,Z 470.975,A -85,B 0,C 180,E1 -22243.122,E2 -22243.122} C_VEL
LIN {X 0,Y 185.72,Z 470.973,A -85,B 0,C 180,E1 -22247.622,E2 -22247.622} C_VEL
LIN {X 0,Y 185.603,Z 470.989,A -85,B 0,C 180,E1 -22252.25,E2 -22252.25} C_VEL
LIN {X 0,Y 185.563,Z 470.996,A -85,B 0,C 180,E1 -22257.031,E2 -22257.031} C_VEL
LIN {X 0,Y 185.574,Z 470.995,A -85,B 0,C 180,E1 -22259.493,E2 -22259.493} C_VEL
LIN {X 0,Y 185.323,Z 471.026,A -85,B 0,C 180,E1 -22264.834,E2 -22264.834} C_VEL
LIN {X 0,Y 190.708,Z 487.377,A -85,B 0,C 180,E1 -22267.234,E2 -22267.234} C_VEL
LIN {X 0,Y 193.746,Z 498.177,A -85,B 0,C 180,E1 -22268.985,E2 -22268.985} C_VEL
LIN {X 0,Y 196.233,Z 509.919,A -85,B 0,C 180,E1 -22271.051,E2 -22271.051} C_VEL
LIN {X 0,Y 197.299,Z 515.985,A -85,B 0,C 180,E1 -22272.214,E2 -22272.214} C_VEL
LIN {X 0,Y 194.828,Z 528.568,A -85,B 0,C 180,E1 -22274.565,E2 -22274.565} C_VEL
LIN {X 0,Y 191.983,Z 541.301,A -85,B 0,C 180,E1 -22277.498,E2 -22277.498} C_VEL
LIN {X 0,Y 189.733,Z 551.15,A -85,B 0,C 180,E1 -22280.285,E2 -22280.285} C_VEL
LIN {X 0,Y 187.419,Z 561.322,A -85,B 0,C 180,E1 -22283.799,E2 -22283.799} C_VEL
LIN {X 0,Y 185.847,Z 569.053,A -85,B 0,C 180,E1 -22287.043,E2 -22287.043} C_VEL
LIN {X 0,Y 184.695,Z 575.617,A -85,B 0,C 180,E1 -22290.351,E2 -22290.351} C_VEL
LIN {X 0,Y 183.807,Z 581.401,A -85,B 0,C 180,E1 -22293.914,E2 -22293.914} C_VEL
LIN {X 0,Y 183.29,Z 585.981,A -85,B 0,C 180,E1 -22297.453,E2 -22297.453} C_VEL
LIN {X 0,Y 183.07,Z 590.591,A -85,B 0,C 180,E1 -22302.114,E2 -22302.114} C_VEL
LIN {X 0,Y 183.279,Z 592.294,A -85,B 0,C 180,E1 -22304.429,E2 -22304.429} C_VEL
LIN {X 0,Y 184.126,Z 594.6,A -85,B 0,C 180,E1 -22308.997,E2 -22308.997} C_VEL
LIN {X 0,Y 185.844,Z 595.571,A -85,B 0,C 180,E1 -22313.485,E2 -22313.485} C_VEL
LIN {X 0,Y 188.445,Z 595.26,A -85,B 0,C 180,E1 -22317.862,E2 -22317.862} C_VEL
LIN {X 0,Y 191.958,Z 593.729,A -85,B 0,C 180,E1 -22322.098,E2 -22322.098} C_VEL
LIN {X 0,Y 196.534,Z 590.912,A -85,B 0,C 180,E1 -22326.158,E2 -22326.158} C_VEL
LIN {X 0,Y 201.991,Z 586.857,A -85,B 0,C 180,E1 -22330.018,E2 -22330.018} C_VEL
LIN {X 0,Y 208.492,Z 581.34,A -85,B 0,C 180,E1 -22333.648,E2 -22333.648} C_VEL
LIN {X 0,Y 215.859,Z 574.359,A -85,B 0,C 180,E1 -22337.039,E2 -22337.039} C_VEL
LIN {X 0,Y 224.042,Z 565.589,A -85,B 0,C 180,E1 -22340.185,E2 -22340.185} C_VEL
LIN {X 0,Y 231.489,Z 556.566,A -85,B 0,C 180,E1 -22342.701,E2 -22342.701} C_VEL
LIN {X 0,Y 232.328,Z 553.18,A -85,B 0,C 180,E1 -22345.056,E2 -22345.056} C_VEL
LIN {X 0,Y 232.484,Z 551.194,A -85,B 0,C 180,E1 -22346.965,E2 -22346.965} C_VEL
LIN {X 0,Y 232.373,Z 549.885,A -85,B 0,C 180,E1 -22348.941,E2 -22348.941} C_VEL
LIN {X 0,Y 232.2,Z 548.742,A -85,B 0,C 180,E1 -22352.064,E2 -22352.064} C_VEL
LIN {X 0,Y 231.939,Z 549.078,A -85,B 0,C 180,E1 -22355.15,E2 -22355.15} C_VEL
LIN {X 0,Y 231.675,Z 550.6,A -85,B 0,C 180,E1 -22357.935,E2 -22357.935} C_VEL
LIN {X 0,Y 231.356,Z 553.147,A -85,B 0,C 180,E1 -22360.587,E2 -22360.587} C_VEL
LIN {X 0,Y 231.052,Z 555.069,A -85,B 0,C 180,E1 -22362.004,E2 -22362.004} C_VEL
LIN {X 0,Y 230.022,Z 557.979,A -85,B 0,C 180,E1 -22363.547,E2 -22363.547} C_VEL
LIN {X 0,Y 227.598,Z 563.764,A -85,B 0,C 180,E1 -22366.005,E2 -22366.005} C_VEL
LIN {X 0,Y 224.458,Z 569.91,A -85,B 0,C 180,E1 -22368.291,E2 -22368.291} C_VEL
LIN {X 0,Y 221.838,Z 574.211,A -85,B 0,C 180,E1 -22369.773,E2 -22369.773} C_VEL
LIN {X 0,Y 213.045,Z 584.642,A -85,B 0,C 180,E1 -22372.985,E2 -22372.985} C_VEL
LIN {X 0,Y 208.226,Z 589.836,A -85,B 0,C 180,E1 -22374.986,E2 -22374.986} C_VEL
LIN {X 0,Y 203.178,Z 595.289,A -85,B 0,C 180,E1 -22377.579,E2 -22377.579} C_VEL
LIN {X 0,Y 197.209,Z 601.397,A -85,B 0,C 180,E1 -22381.243,E2 -22381.243} C_VEL
LIN {X 0,Y 192.257,Z 606.21,A -85,B 0,C 180,E1 -22385.142,E2 -22385.142} C_VEL
LIN {X 0,Y 189.233,Z 609.022,A -85,B 0,C 180,E1 -22388.199,E2 -22388.199} C_VEL
LIN {X 0,Y 186.244,Z 611.783,A -85,B 0,C 180,E1 -22392.43,E2 -22392.43} C_VEL
LIN {X 0,Y 184.267,Z 613.403,A -85,B 0,C 180,E1 -22396.771,E2 -22396.771} C_VEL
LIN {X 0,Y 183.421,Z 613.86,A -85,B 0,C 180,E1 -22401.184,E2 -22401.184} C_VEL
LIN {X 0,Y 183.394,Z 613.331,A -85,B 0,C 180,E1 -22404.692,E2 -22404.692} C_VEL
LIN {X 0,Y 182.83,Z 612.69,A -85,B 0,C 180,E1 -22406.516,E2 -22406.516} C_VEL
LIN {X 0,Y 181.309,Z 611.694,A -85,B 0,C 180,E1 -22408.299,E2 -22408.299} C_VEL
LIN {X 0,Y 177.687,Z 608.82,A -85,B 0,C 180,E1 -22411.859,E2 -22411.859} C_VEL
LIN {X 0,Y 176.737,Z 607.086,A -85,B 0,C 180,E1 -22413.7,E2 -22413.7} C_VEL
LIN {X 0,Y 176.699,Z 606.448,A -85,B 0,C 180,E1 -22414.32,E2 -22414.32} C_VEL
LIN {X 0,Y 176.789,Z 602.26,A -85,B 0,C 180,E1 -22417.998,E2 -22417.998} C_VEL
LIN {X 0,Y 177.172,Z 597.267,A -85,B 0,C 180,E1 -22421.44,E2 -22421.44} C_VEL
LIN {X 0,Y 178.122,Z 590.016,A -85,B 0,C 180,E1 -22425.446,E2 -22425.446} C_VEL
LIN {X 0,Y 179.891,Z 581.024,A -85,B 0,C 180,E1 -22429.395,E2 -22429.395} C_VEL
LIN {X 0,Y 182.003,Z 571.702,A -85,B 0,C 180,E1 -22432.715,E2 -22432.715} C_VEL
LIN {X 0,Y 184.675,Z 560.499,A -85,B 0,C 180,E1 -22435.953,E2 -22435.953} C_VEL
LIN {X 0,Y 186.891,Z 550.419,A -85,B 0,C 180,E1 -22438.343,E2 -22438.343} C_VEL
LIN {X 0,Y 186.13,Z 537.595,A -85,B 0,C 180,E1 -22441.071,E2 -22441.071} C_VEL
LIN {X 0,Y 185.182,Z 524.748,A -85,B 0,C 180,E1 -22443.391,E2 -22443.391} C_VEL
LIN {X 0,Y 183.685,Z 510.391,A -85,B 0,C 180,E1 -22445.581,E2 -22445.581} C_VEL
LIN {X 0,Y 181.627,Z 494.229,A -85,B 0,C 180,E1 -22447.607,E2 -22447.607} C_VEL
LIN {X 0,Y 180.282,Z 485.05,A -85,B 0,C 180,E1 -22448.588,E2 -22448.588} C_VEL
LIN {X 0,Y 180.561,Z 482.668,A -85,B 0,C 180,E1 -22451.428,E2 -22451.428} C_VEL
LIN {X 0,Y 180.086,Z 479.488,A -85,B 0,C 180,E1 -22455.375,E2 -22455.375} C_VEL
LIN {X 0,Y 179.372,Z 476.147,A -85,B 0,C 180,E1 -22459.723,E2 -22459.723} C_VEL
LIN {X 0,Y 178.639,Z 471.854,A -85,B 0,C 180,E1 -22465.707,E2 -22465.707} C_VEL
LIN {X 0,Y 178.523,Z 471.873,A -85,B 0,C 180,E1 -22470.005,E2 -22470.005} C_VEL
LIN {X 0,Y 178.532,Z 471.864,A -85,B 0,C 180,E1 -22474.876,E2 -22474.876} C_VEL
LIN {X 0,Y 178.636,Z 471.86,A -85,B 0,C 180,E1 -22480.77,E2 -22480.77} C_VEL
LIN {X 0,Y 178.672,Z 471.848,A -85,B 0,C 180,E1 -22484.018,E2 -22484.018} C_VEL
LIN {X 0,Y 178.859,Z 471.83,A -85,B 0,C 180,E1 -22489.21,E2 -22489.21} C_VEL
LIN {X 0,Y 178.922,Z 471.818,A -85,B 0,C 180,E1 -22493.233,E2 -22493.233} C_VEL
LIN {X 0,Y 179.151,Z 471.793,A -85,B 0,C 180,E1 -22497.752,E2 -22497.752} C_VEL
LIN {X 0,Y 179.367,Z 471.765,A -85,B 0,C 180,E1 -22500,E2 -22500} C_VEL
LIN {X 0,Y 178.874,Z 471.828,A -85,B 0,C 180,E1 -22504.507,E2 -22504.507} C_VEL
LIN {X 0,Y 178.958,Z 471.814,A -85,B 0,C 180,E1 -22509.038,E2 -22509.038} C_VEL
LIN {X 0,Y 178.679,Z 471.851,A -85,B 0,C 180,E1 -22513.651,E2 -22513.651} C_VEL
LIN {X 0,Y 178.622,Z 471.853,A -85,B 0,C 180,E1 -22519.217,E2 -22519.217} C_VEL
LIN {X 0,Y 178.533,Z 471.869,A -85,B 0,C 180,E1 -22525.125,E2 -22525.125} C_VEL
LIN {X 0,Y 178.478,Z 471.876,A -85,B 0,C 180,E1 -22530.791,E2 -22530.791} C_VEL
LIN {X 0,Y 178.495,Z 471.875,A -85,B 0,C 180,E1 -22534.226,E2 -22534.226} C_VEL
LIN {X 0,Y 178.418,Z 471.883,A -85,B 0,C 180,E1 -22539.069,E2 -22539.069} C_VEL
LIN {X 0,Y 178.412,Z 471.887,A -85,B 0,C 180,E1 -22542.042,E2 -22542.042} C_VEL
LIN {X 0,Y 178.419,Z 471.88,A -85,B 0,C 180,E1 -22545.157,E2 -22545.157} C_VEL
LIN {X 0,Y 178.426,Z 471.883,A -85,B 0,C 180,E1 -22548.452,E2 -22548.452} C_VEL
LIN {X 0,Y 178.451,Z 471.878,A -85,B 0,C 180,E1 -22553.79,E2 -22553.79} C_VEL
LIN {X 0,Y 178.493,Z 471.874,A -85,B 0,C 180,E1 -22556.549,E2 -22556.549} C_VEL
LIN {X 0,Y 178.525,Z 471.872,A -85,B 0,C 180,E1 -22560.007,E2 -22560.007} C_VEL
LIN {X 0,Y 178.537,Z 471.867,A -85,B 0,C 180,E1 -22564.876,E2 -22564.876} C_VEL
LIN {X 0,Y 178.626,Z 471.856,A -85,B 0,C 180,E1 -22570.784,E2 -22570.784} C_VEL
LIN {X 0,Y 178.661,Z 471.854,A -85,B 0,C 180,E1 -22576.348,E2 -22576.348} C_VEL
LIN {X 0,Y 178.909,Z 471.819,A -85,B 0,C 180,E1 -22580.96,E2 -22580.96} C_VEL
LIN {X 0,Y 179.154,Z 471.791,A -85,B 0,C 180,E1 -22587.752,E2 -22587.752} C_VEL
LIN {X 0,Y 179.373,Z 471.761,A -85,B 0,C 180,E1 -22590,E2 -22590} C_VEL
LIN {X 0,Y 178.873,Z 471.827,A -85,B 0,C 180,E1 -22594.507,E2 -22594.507} C_VEL
LIN {X 0,Y 178.918,Z 471.817,A -85,B 0,C 180,E1 -22599.04,E2 -22599.04} C_VEL
LIN {X 0,Y 178.663,Z 471.856,A -85,B 0,C 180,E1 -22603.651,E2 -22603.651} C_VEL
LIN {X 0,Y 178.641,Z 471.858,A -85,B 0,C 180,E1 -22609.23,E2 -22609.23} C_VEL
LIN {X 0,Y 178.537,Z 471.872,A -85,B 0,C 180,E1 -22615.124,E2 -22615.124} C_VEL
LIN {X 0,Y 178.492,Z 471.877,A -85,B 0,C 180,E1 -22619.975,E2 -22619.975} C_VEL
LIN {X 0,Y 178.32,Z 471.897,A -85,B 0,C 180,E1 -22624.014,E2 -22624.014} C_VEL
LIN {X 0,Y 183.129,Z 486.365,A -85,B 0,C 180,E1 -22626.216,E2 -22626.216} C_VEL
LIN {X 0,Y 186.808,Z 498.988,A -85,B 0,C 180,E1 -22628.37,E2 -22628.37} C_VEL
LIN {X 0,Y 189.476,Z 511.806,A -85,B 0,C 180,E1 -22630.75,E2 -22630.75} C_VEL
LIN {X 0,Y 190.315,Z 517.42,A -85,B 0,C 180,E1 -22631.876,E2 -22631.876} C_VEL
LIN {X 0,Y 187.716,Z 529.692,A -85,B 0,C 180,E1 -22634.271,E2 -22634.271} C_VEL
LIN {X 0,Y 184.916,Z 541.892,A -85,B 0,C 180,E1 -22637.205,E2 -22637.205} C_VEL
LIN {X 0,Y 182.366,Z 552.693,A -85,B 0,C 180,E1 -22640.421,E2 -22640.421} C_VEL
LIN {X 0,Y 180.022,Z 562.887,A -85,B 0,C 180,E1 -22644.154,E2 -22644.154} C_VEL
LIN {X 0,Y 178.379,Z 571.073,A -85,B 0,C 180,E1 -22647.866,E2 -22647.866} C_VEL
LIN {X 0,Y 177.209,Z 577.756,A -85,B 0,C 180,E1 -22651.581,E2 -22651.581} C_VEL
LIN {X 0,Y 176.444,Z 583.178,A -85,B 0,C 180,E1 -22655.278,E2 -22655.278} C_VEL
LIN {X 0,Y 176.04,Z 587.515,A -85,B 0,C 180,E1 -22658.942,E2 -22658.942} C_VEL
LIN {X 0,Y 176.105,Z 591.759,A -85,B 0,C 180,E1 -22663.778,E2 -22663.778} C_VEL
LIN {X 0,Y 176.881,Z 594.504,A -85,B 0,C 180,E1 -22668.541,E2 -22668.541} C_VEL
LIN {X 0,Y 178.573,Z 595.912,A -85,B 0,C 180,E1 -22673.219,E2 -22673.219} C_VEL
LIN {X 0,Y 181.154,Z 596.038,A -85,B 0,C 180,E1 -22677.776,E2 -22677.776} C_VEL
LIN {X 0,Y 184.719,Z 594.932,A -85,B 0,C 180,E1 -22682.18,E2 -22682.18} C_VEL
LIN {X 0,Y 189.373,Z 592.6,A -85,B 0,C 180,E1 -22686.392,E2 -22686.392} C_VEL
LIN {X 0,Y 194.958,Z 589.013,A -85,B 0,C 180,E1 -22690.384,E2 -22690.384} C_VEL
LIN {X 0,Y 201.615,Z 584.085,A -85,B 0,C 180,E1 -22694.123,E2 -22694.123} C_VEL
LIN {X 0,Y 209.137,Z 577.68,A -85,B 0,C 180,E1 -22697.604,E2 -22697.604} C_VEL
LIN {X 0,Y 217.561,Z 569.622,A -85,B 0,C 180,E1 -22700.814,E2 -22700.814} C_VEL
LIN {X 0,Y 225.494,Z 561.024,A -85,B 0,C 180,E1 -22703.414,E2 -22703.414} C_VEL
LIN {X 0,Y 226.44,Z 559.862,A -85,B 0,C 180,E1 -22703.796,E2 -22703.796} C_VEL
LIN {X 0,Y 227.143,Z 557.519,A -85,B 0,C 180,E1 -22705.669,E2 -22705.669} C_VEL
LIN {X 0,Y 227.428,Z 555.832,A -85,B 0,C 180,E1 -22707.615,E2 -22707.615} C_VEL
LIN {X 0,Y 227.384,Z 554.549,A -85,B 0,C 180,E1 -22710.071,E2 -22710.071} C_VEL
LIN {X 0,Y 227.394,Z 554.038,A -85,B 0,C 180,E1 -22711.696,E2 -22711.696} C_VEL
LIN {X 0,Y 227.25,Z 554.079,A -85,B 0,C 180,E1 -22713.826,E2 -22713.826} C_VEL
LIN {X 0,Y 226.968,Z 554.975,A -85,B 0,C 180,E1 -22716.383,E2 -22716.383} C_VEL
LIN {X 0,Y 226.602,Z 556.945,A -85,B 0,C 180,E1 -22719.163,E2 -22719.163} C_VEL
LIN {X 0,Y 226.202,Z 558.646,A -85,B 0,C 180,E1 -22720.727,E2 -22720.727} C_VEL
LIN {X 0,Y 225.441,Z 560.973,A -85,B 0,C 180,E1 -22722.268,E2 -22722.268} C_VEL
LIN {X 0,Y 223.001,Z 565.945,A -85,B 0,C 180,E1 -22724.625,E2 -22724.625} C_VEL
LIN {X 0,Y 219.428,Z 572.102,A -85,B 0,C 180,E1 -22727.11,E2 -22727.11} C_VEL
LIN {X 0,Y 217.03,Z 575.686,A -85,B 0,C 180,E1 -22728.431,E2 -22728.431} C_VEL
LIN {X 0,Y 208.544,Z 584.989,A -85,B 0,C 180,E1 -22731.432,E2 -22731.432} C_VEL
LIN {X 0,Y 202.531,Z 591.008,A -85,B 0,C 180,E1 -22733.85,E2 -22733.85} C_VEL
LIN {X 0,Y 197.277,Z 596.164,A -85,B 0,C 180,E1 -22736.483,E2 -22736.483} C_VEL
LIN {X 0,Y 191.036,Z 601.916,A -85,B 0,C 180,E1 -22740.222,E2 -22740.222} C_VEL
LIN {X 0,Y 187.054,Z 605.444,A -85,B 0,C 180,E1 -22743.201,E2 -22743.201} C_VEL
LIN {X 0,Y 182.369,Z 609.308,A -85,B 0,C 180,E1 -22747.652,E2 -22747.652} C_VEL
LIN {X 0,Y 179.434,Z 611.612,A -85,B 0,C 180,E1 -22751.74,E2 -22751.74} C_VEL
LIN {X 0,Y 177.314,Z 613.005,A -85,B 0,C 180,E1 -22756.243,E2 -22756.243} C_VEL
LIN {X 0,Y 176.403,Z 613.254,A -85,B 0,C 180,E1 -22760.83,E2 -22760.83} C_VEL
LIN {X 0,Y 176.437,Z 612.32,A -85,B 0,C 180,E1 -22765.431,E2 -22765.431} C_VEL
LIN {X 0,Y 176.778,Z 610.046,A -85,B 0,C 180,E1 -22770,E2 -22770} C_VEL
LIN {X 0,Y 176.699,Z 606.448,A -85,B 0,C 180,E1 -22774.32,E2 -22774.32} C_VEL
LIN {X 0,Y 176.147,Z 604.474,A -85,B 0,C 180,E1 -22776.109,E2 -22776.109} C_VEL
LIN {X 0,Y 174.662,Z 602.184,A -85,B 0,C 180,E1 -22777.833,E2 -22777.833} C_VEL
LIN {X 0,Y 170.886,Z 595.954,A -85,B 0,C 180,E1 -22781.802,E2 -22781.802} C_VEL
LIN {X 0,Y 170.575,Z 592.973,A -85,B 0,C 180,E1 -22783.539,E2 -22783.539} C_VEL
LIN {X 0,Y 171.719,Z 585.788,A -85,B 0,C 180,E1 -22787.261,E2 -22787.261} C_VEL
LIN {X 0,Y 173.501,Z 577.517,A -85,B 0,C 180,E1 -22790.758,E2 -22790.758} C_VEL
LIN {X 0,Y 175.846,Z 567.565,A -85,B 0,C 180,E1 -22794.183,E2 -22794.183} C_VEL
LIN {X 0,Y 178.8,Z 555.555,A -85,B 0,C 180,E1 -22797.506,E2 -22797.506} C_VEL
LIN {X 0,Y 179.826,Z 550.943,A -85,B 0,C 180,E1 -22798.604,E2 -22798.604} C_VEL
LIN {X 0,Y 179.216,Z 538.934,A -85,B 0,C 180,E1 -22801.305,E2 -22801.305} C_VEL
LIN {X 0,Y 178.258,Z 525.317,A -85,B 0,C 180,E1 -22803.917,E2 -22803.917} C_VEL
LIN {X 0,Y 176.899,Z 511.281,A -85,B 0,C 180,E1 -22806.199,E2 -22806.199} C_VEL
LIN {X 0,Y 175.058,Z 496.15,A -85,B 0,C 180,E1 -22808.207,E2 -22808.207} C_VEL
LIN {X 0,Y 173.314,Z 484.658,A -85,B 0,C 180,E1 -22809.525,E2 -22809.525} C_VEL
LIN {X 0,Y 173.465,Z 482.902,A -85,B 0,C 180,E1 -22811.72,E2 -22811.72} C_VEL
LIN {X 0,Y 172.866,Z 479.411,A -85,B 0,C 180,E1 -22816.28,E2 -22816.28} C_VEL
LIN {X 0,Y 172.13,Z 476.038,A -85,B 0,C 180,E1 -22820.873,E2 -22820.873} C_VEL
LIN {X 0,Y 171.588,Z 472.732,A -85,B 0,C 180,E1 -22825.724,E2 -22825.724} C_VEL
LIN {X 0,Y 171.449,Z 472.755,A -85,B 0,C 180,E1 -22830.535,E2 -22830.535} C_VEL
LIN {X 0,Y 171.456,Z 472.747,A -85,B 0,C 180,E1 -22835.802,E2 -22835.802} C_VEL
LIN {X 0,Y 171.593,Z 472.736,A -85,B 0,C 180,E1 -22840.874,E2 -22840.874} C_VEL
LIN {X 0,Y 171.61,Z 472.73,A -85,B 0,C 180,E1 -22845.776,E2 -22845.776} C_VEL
LIN {X 0,Y 171.886,Z 472.699,A -85,B 0,C 180,E1 -22850.587,E2 -22850.587} C_VEL
LIN {X 0,Y 171.82,Z 472.705,A -85,B 0,C 180,E1 -22855.308,E2 -22855.308} C_VEL
LIN {X 0,Y 172.33,Z 472.642,A -85,B 0,C 180,E1 -22860,E2 -22860} C_VEL
LIN {X 0,Y 171.823,Z 472.708,A -85,B 0,C 180,E1 -22864.693,E2 -22864.693} C_VEL
LIN {X 0,Y 171.887,Z 472.695,A -85,B 0,C 180,E1 -22869.413,E2 -22869.413} C_VEL
LIN {X 0,Y 171.592,Z 472.736,A -85,B 0,C 180,E1 -22874.226,E2 -22874.226} C_VEL
LIN {X 0,Y 171.543,Z 472.735,A -85,B 0,C 180,E1 -22879.562,E2 -22879.562} C_VEL
LIN {X 0,Y 171.468,Z 472.75,A -85,B 0,C 180,E1 -22885.617,E2 -22885.617} C_VEL
LIN {X 0,Y 171.441,Z 472.754,A -85,B 0,C 180,E1 -22890.588,E2 -22890.588} C_VEL
LIN {X 0,Y 171.406,Z 472.756,A -85,B 0,C 180,E1 -22895.032,E2 -22895.032} C_VEL
LIN {X 0,Y 171.379,Z 472.759,A -85,B 0,C 180,E1 -22898.818,E2 -22898.818} C_VEL
LIN {X 0,Y 171.34,Z 472.764,A -85,B 0,C 180,E1 -22904.212,E2 -22904.212} C_VEL
LIN {X 0,Y 171.357,Z 472.763,A -85,B 0,C 180,E1 -22908.989,E2 -22908.989} C_VEL
LIN {X 0,Y 171.416,Z 472.757,A -85,B 0,C 180,E1 -22912.049,E2 -22912.049} C_VEL
LIN {X 0,Y 171.412,Z 472.752,A -85,B 0,C 180,E1 -22915.087,E2 -22915.087} C_VEL
LIN {X 0,Y 171.451,Z 472.751,A -85,B 0,C 180,E1 -22920.535,E2 -22920.535} C_VEL
LIN {X 0,Y 171.46,Z 472.752,A -85,B 0,C 180,E1 -22925.802,E2 -22925.802} C_VEL
LIN {X 0,Y 171.582,Z 472.733,A -85,B 0,C 180,E1 -22930.872,E2 -22930.872} C_VEL
LIN {X 0,Y 171.579,Z 472.738,A -85,B 0,C 180,E1 -22935.773,E2 -22935.773} C_VEL
LIN {X 0,Y 171.847,Z 472.698,A -85,B 0,C 180,E1 -22940.585,E2 -22940.585} C_VEL
LIN {X 0,Y 171.813,Z 472.709,A -85,B 0,C 180,E1 -22945.307,E2 -22945.307} C_VEL
LIN {X 0,Y 172.336,Z 472.638,A -85,B 0,C 180,E1 -22950,E2 -22950} C_VEL
LIN {X 0,Y 171.822,Z 472.706,A -85,B 0,C 180,E1 -22954.692,E2 -22954.692} C_VEL
LIN {X 0,Y 171.853,Z 472.696,A -85,B 0,C 180,E1 -22959.415,E2 -22959.415} C_VEL
LIN {X 0,Y 171.583,Z 472.737,A -85,B 0,C 180,E1 -22964.226,E2 -22964.226} C_VEL
LIN {X 0,Y 171.56,Z 472.741,A -85,B 0,C 180,E1 -22969.574,E2 -22969.574} C_VEL
LIN {X 0,Y 171.471,Z 472.75,A -85,B 0,C 180,E1 -22975.616,E2 -22975.616} C_VEL
LIN {X 0,Y 171.403,Z 472.761,A -85,B 0,C 180,E1 -22980.563,E2 -22980.563} C_VEL
LIN {X 0,Y 171.322,Z 472.891,A -85,B 0,C 180,E1 -22983.187,E2 -22983.187} C_VEL
LIN {X 0,Y 176.437,Z 488.146,A -85,B 0,C 180,E1 -22985.638,E2 -22985.638} C_VEL
LIN {X 0,Y 180.094,Z 500.726,A -85,B 0,C 180,E1 -22987.885,E2 -22987.885} C_VEL
LIN {X 0,Y 182.684,Z 513.532,A -85,B 0,C 180,E1 -22990.395,E2 -22990.395} C_VEL
LIN {X 0,Y 183.38,Z 517.795,A -85,B 0,C 180,E1 -22991.305,E2 -22991.305} C_VEL
LIN {X 0,Y 180.745,Z 530.219,A -85,B 0,C 180,E1 -22993.824,E2 -22993.824} C_VEL
LIN {X 0,Y 178.015,Z 541.747,A -85,B 0,C 180,E1 -22996.688,E2 -22996.688} C_VEL
LIN {X 0,Y 175.316,Z 552.819,A -85,B 0,C 180,E1 -23000.103,E2 -23000.103} C_VEL
LIN {X 0,Y 173.092,Z 562.224,A -85,B 0,C 180,E1 -23003.656,E2 -23003.656} C_VEL
LIN {X 0,Y 171.301,Z 571.077,A -85,B 0,C 180,E1 -23007.767,E2 -23007.767} C_VEL
LIN {X 0,Y 170.076,Z 577.835,A -85,B 0,C 180,E1 -23011.626,E2 -23011.626} C_VEL
LIN {X 0,Y 169.263,Z 583.98,A -85,B 0,C 180,E1 -23015.986,E2 -23015.986} C_VEL
LIN {X 0,Y 168.875,Z 588.918,A -85,B 0,C 180,E1 -23020.553,E2 -23020.553} C_VEL
LIN {X 0,Y 169.201,Z 592.874,A -85,B 0,C 180,E1 -23025.568,E2 -23025.568} C_VEL
LIN {X 0,Y 170.347,Z 595.39,A -85,B 0,C 180,E1 -23030.501,E2 -23030.501} C_VEL
LIN {X 0,Y 172.423,Z 596.582,A -85,B 0,C 180,E1 -23035.324,E2 -23035.324} C_VEL
LIN {X 0,Y 175.698,Z 596.491,A -85,B 0,C 180,E1 -23040.197,E2 -23040.197} C_VEL
LIN {X 0,Y 179.699,Z 595.251,A -85,B 0,C 180,E1 -23044.486,E2 -23044.486} C_VEL
LIN {X 0,Y 184.962,Z 592.746,A -85,B 0,C 180,E1 -23048.742,E2 -23048.742} C_VEL
LIN {X 0,Y 191.184,Z 589.036,A -85,B 0,C 180,E1 -23052.742,E2 -23052.742} C_VEL
LIN {X 0,Y 198.476,Z 583.909,A -85,B 0,C 180,E1 -23056.456,E2 -23056.456} C_VEL
LIN {X 0,Y 206.649,Z 577.345,A -85,B 0,C 180,E1 -23059.882,E2 -23059.882} C_VEL
LIN {X 0,Y 215.623,Z 569.141,A -85,B 0,C 180,E1 -23063.024,E2 -23063.024} C_VEL
LIN {X 0,Y 220.404,Z 564.352,A -85,B 0,C 180,E1 -23064.489,E2 -23064.489} C_VEL
LIN {X 0,Y 221.569,Z 562.706,A -85,B 0,C 180,E1 -23065.354,E2 -23065.354} C_VEL
LIN {X 0,Y 222.168,Z 560.724,A -85,B 0,C 180,E1 -23067.659,E2 -23067.659} C_VEL
LIN {X 0,Y 222.332,Z 559.14,A -85,B 0,C 180,E1 -23071.41,E2 -23071.41} C_VEL
LIN {X 0,Y 222.303,Z 559.023,A -85,B 0,C 180,E1 -23072.51,E2 -23072.51} C_VEL
LIN {X 0,Y 222.083,Z 559.389,A -85,B 0,C 180,E1 -23074.724,E2 -23074.724} C_VEL
LIN {X 0,Y 221.704,Z 560.78,A -85,B 0,C 180,E1 -23077.582,E2 -23077.582} C_VEL
LIN {X 0,Y 221.057,Z 563.197,A -85,B 0,C 180,E1 -23080.27,E2 -23080.27} C_VEL
LIN {X 0,Y 220.328,Z 564.918,A -85,B 0,C 180,E1 -23081.515,E2 -23081.515} C_VEL
LIN {X 0,Y 217.618,Z 569.59,A -85,B 0,C 180,E1 -23083.848,E2 -23083.848} C_VEL
LIN {X 0,Y 213.703,Z 575.386,A -85,B 0,C 180,E1 -23086.322,E2 -23086.322} C_VEL
LIN {X 0,Y 211.972,Z 577.613,A -85,B 0,C 180,E1 -23087.207,E2 -23087.207} C_VEL
LIN {X 0,Y 203.15,Z 586.457,A -85,B 0,C 180,E1 -23090.208,E2 -23090.208} C_VEL
LIN {X 0,Y 196.917,Z 592.146,A -85,B 0,C 180,E1 -23092.647,E2 -23092.647} C_VEL
LIN {X 0,Y 191.454,Z 597.035,A -85,B 0,C 180,E1 -23095.321,E2 -23095.321} C_VEL
LIN {X 0,Y 184.932,Z 602.46,A -85,B 0,C 180,E1 -23099.134,E2 -23099.134} C_VEL
LIN {X 0,Y 178.239,Z 607.589,A -85,B 0,C 180,E1 -23104.296,E2 -23104.296} C_VEL
LIN {X 0,Y 174.239,Z 610.431,A -85,B 0,C 180,E1 -23108.715,E2 -23108.715} C_VEL
LIN {X 0,Y 171.38,Z 612.173,A -85,B 0,C 180,E1 -23113.318,E2 -23113.318} C_VEL
LIN {X 0,Y 169.757,Z 612.775,A -85,B 0,C 180,E1 -23118.053,E2 -23118.053} C_VEL
LIN {X 0,Y 169.255,Z 612.227,A -85,B 0,C 180,E1 -23122.844,E2 -23122.844} C_VEL
LIN {X 0,Y 169.384,Z 611.512,A -85,B 0,C 180,E1 -23125.24,E2 -23125.24} C_VEL
LIN {X 0,Y 169.752,Z 609.07,A -85,B 0,C 180,E1 -23130,E2 -23130} C_VEL
LIN {X 0,Y 169.68,Z 605.019,A -85,B 0,C 180,E1 -23134.752,E2 -23134.752} C_VEL
LIN {X 0,Y 169.781,Z 600.846,A -85,B 0,C 180,E1 -23138.33,E2 -23138.33} C_VEL
LIN {X 0,Y 170.224,Z 595.681,A -85,B 0,C 180,E1 -23141.913,E2 -23141.913} C_VEL
LIN {X 0,Y 170.575,Z 592.973,A -85,B 0,C 180,E1 -23143.539,E2 -23143.539} C_VEL
LIN {X 0,Y 170.396,Z 589.859,A -85,B 0,C 180,E1 -23145.22,E2 -23145.22} C_VEL
LIN {X 0,Y 168.54,Z 584.171,A -85,B 0,C 180,E1 -23147.893,E2 -23147.893} C_VEL
LIN {X 0,Y 166.91,Z 578.04,A -85,B 0,C 180,E1 -23150.507,E2 -23150.507} C_VEL
LIN {X 0,Y 167.107,Z 574.101,A -85,B 0,C 180,E1 -23152.044,E2 -23152.044} C_VEL
LIN {X 0,Y 169.328,Z 564.953,A -85,B 0,C 180,E1 -23155.177,E2 -23155.177} C_VEL
LIN {X 0,Y 171.935,Z 554.843,A -85,B 0,C 180,E1 -23158.038,E2 -23158.038} C_VEL
LIN {X 0,Y 172.756,Z 551.452,A -85,B 0,C 180,E1 -23158.887,E2 -23158.887} C_VEL
LIN {X 0,Y 172.239,Z 539.37,A -85,B 0,C 180,E1 -23161.736,E2 -23161.736} C_VEL
LIN {X 0,Y 171.303,Z 525.414,A -85,B 0,C 180,E1 -23164.534,E2 -23164.534} C_VEL
LIN {X 0,Y 170.046,Z 511.537,A -85,B 0,C 180,E1 -23166.885,E2 -23166.885} C_VEL
LIN {X 0,Y 168.207,Z 496.139,A -85,B 0,C 180,E1 -23169.048,E2 -23169.048} C_VEL
LIN {X 0,Y 166.345,Z 484.296,A -85,B 0,C 180,E1 -23170.493,E2 -23170.493} C_VEL
LIN {X 0,Y 166.092,Z 481.656,A -85,B 0,C 180,E1 -23174.001,E2 -23174.001} C_VEL
LIN {X 0,Y 165.616,Z 479.309,A -85,B 0,C 180,E1 -23177.238,E2 -23177.238} C_VEL
LIN {X 0,Y 164.925,Z 476.123,A -85,B 0,C 180,E1 -23181.838,E2 -23181.838} C_VEL
LIN {X 0,Y 164.542,Z 473.61,A -85,B 0,C 180,E1 -23185.743,E2 -23185.743} C_VEL
LIN {X 0,Y 164.418,Z 473.632,A -85,B 0,C 180,E1 -23189.141,E2 -23189.141} C_VEL
LIN {X 0,Y 164.414,Z 473.622,A -85,B 0,C 180,E1 -23194.694,E2 -23194.694} C_VEL
LIN {X 0,Y 164.484,Z 473.62,A -85,B 0,C 180,E1 -23200.05,E2 -23200.05} C_VEL
LIN {X 0,Y 164.556,Z 473.609,A -85,B 0,C 180,E1 -23205.153,E2 -23205.153} C_VEL
LIN {X 0,Y 164.806,Z 473.58,A -85,B 0,C 180,E1 -23210.179,E2 -23210.179} C_VEL
LIN {X 0,Y 164.849,Z 473.571,A -85,B 0,C 180,E1 -23212.652,E2 -23212.652} C_VEL
LIN {X 0,Y 165.048,Z 473.55,A -85,B 0,C 180,E1 -23217.56,E2 -23217.56} C_VEL
LIN {X 0,Y 165.293,Z 473.518,A -85,B 0,C 180,E1 -23220,E2 -23220} C_VEL
LIN {X 0,Y 164.773,Z 473.585,A -85,B 0,C 180,E1 -23224.894,E2 -23224.894} C_VEL
LIN {X 0,Y 164.85,Z 473.574,A -85,B 0,C 180,E1 -23227.349,E2 -23227.349} C_VEL
LIN {X 0,Y 164.752,Z 473.583,A -85,B 0,C 180,E1 -23231.152,E2 -23231.152} C_VEL
LIN {X 0,Y 164.483,Z 473.618,A -85,B 0,C 180,E1 -23237.404,E2 -23237.404} C_VEL
LIN {X 0,Y 164.472,Z 473.617,A -85,B 0,C 180,E1 -23239.99,E2 -23239.99} C_VEL
LIN {X 0,Y 164.393,Z 473.631,A -85,B 0,C 180,E1 -23246.135,E2 -23246.135} C_VEL
LIN {X 0,Y 164.375,Z 473.633,A -85,B 0,C 180,E1 -23251.229,E2 -23251.229} C_VEL
LIN {X 0,Y 164.312,Z 473.636,A -85,B 0,C 180,E1 -23256.786,E2 -23256.786} C_VEL
LIN {X 0,Y 164.3,Z 473.643,A -85,B 0,C 180,E1 -23259.914,E2 -23259.914} C_VEL
LIN {X 0,Y 164.279,Z 473.645,A -85,B 0,C 180,E1 -23263.343,E2 -23263.343} C_VEL
LIN {X 0,Y 164.293,Z 473.64,A -85,B 0,C 180,E1 -23266.81,E2 -23266.81} C_VEL
LIN {X 0,Y 164.31,Z 473.643,A -85,B 0,C 180,E1 -23270.347,E2 -23270.347} C_VEL
LIN {X 0,Y 164.344,Z 473.632,A -85,B 0,C 180,E1 -23274.343,E2 -23274.343} C_VEL
LIN {X 0,Y 164.393,Z 473.632,A -85,B 0,C 180,E1 -23279.136,E2 -23279.136} C_VEL
LIN {X 0,Y 164.419,Z 473.625,A -85,B 0,C 180,E1 -23284.695,E2 -23284.695} C_VEL
LIN {X 0,Y 164.487,Z 473.618,A -85,B 0,C 180,E1 -23290.052,E2 -23290.052} C_VEL
LIN {X 0,Y 164.527,Z 473.614,A -85,B 0,C 180,E1 -23295.15,E2 -23295.15} C_VEL
LIN {X 0,Y 164.768,Z 473.58,A -85,B 0,C 180,E1 -23300.177,E2 -23300.177} C_VEL
LIN {X 0,Y 164.829,Z 473.574,A -85,B 0,C 180,E1 -23302.651,E2 -23302.651} C_VEL
LIN {X 0,Y 165.049,Z 473.549,A -85,B 0,C 180,E1 -23307.56,E2 -23307.56} C_VEL
LIN {X 0,Y 165.298,Z 473.514,A -85,B 0,C 180,E1 -23310,E2 -23310} C_VEL
LIN {X 0,Y 164.771,Z 473.585,A -85,B 0,C 180,E1 -23314.894,E2 -23314.894} C_VEL
LIN {X 0,Y 164.838,Z 473.573,A -85,B 0,C 180,E1 -23317.349,E2 -23317.349} C_VEL
LIN {X 0,Y 164.706,Z 473.588,A -85,B 0,C 180,E1 -23321.062,E2 -23321.062} C_VEL
LIN {X 0,Y 164.501,Z 473.616,A -85,B 0,C 180,E1 -23327.401,E2 -23327.401} C_VEL
LIN {X 0,Y 164.478,Z 473.622,A -85,B 0,C 180,E1 -23329.988,E2 -23329.988} C_VEL
LIN {X 0,Y 164.395,Z 473.631,A -85,B 0,C 180,E1 -23336.133,E2 -23336.133} C_VEL
LIN {X 0,Y 164.275,Z 473.648,A -85,B 0,C 180,E1 -23342.179,E2 -23342.179} C_VEL
LIN {X 0,Y 169.759,Z 490.105,A -85,B 0,C 180,E1 -23345.059,E2 -23345.059} C_VEL
LIN {X 0,Y 173.373,Z 502.623,A -85,B 0,C 180,E1 -23347.448,E2 -23347.448} C_VEL
LIN {X 0,Y 175.826,Z 514.892,A -85,B 0,C 180,E1 -23349.977,E2 -23349.977} C_VEL
LIN {X 0,Y 176.399,Z 518.575,A -85,B 0,C 180,E1 -23350.8,E2 -23350.8} C_VEL
LIN {X 0,Y 173.632,Z 531.155,A -85,B 0,C 180,E1 -23353.479,E2 -23353.479} C_VEL
LIN {X 0,Y 170.826,Z 542.745,A -85,B 0,C 180,E1 -23356.52,E2 -23356.52} C_VEL
LIN {X 0,Y 167.895,Z 554.41,A -85,B 0,C 180,E1 -23360.33,E2 -23360.33} C_VEL
LIN {X 0,Y 165.58,Z 564.213,A -85,B 0,C 180,E1 -23364.294,E2 -23364.294} C_VEL
LIN {X 0,Y 163.981,Z 572.33,A -85,B 0,C 180,E1 -23368.33,E2 -23368.33} C_VEL
LIN {X 0,Y 162.65,Z 579.885,A -85,B 0,C 180,E1 -23373.018,E2 -23373.018} C_VEL
LIN {X 0,Y 162.043,Z 585.009,A -85,B 0,C 180,E1 -23377.024,E2 -23377.024} C_VEL
LIN {X 0,Y 161.791,Z 589.089,A -85,B 0,C 180,E1 -23380.986,E2 -23380.986} C_VEL
LIN {X 0,Y 161.992,Z 592.29,A -85,B 0,C 180,E1 -23384.911,E2 -23384.911} C_VEL
LIN {X 0,Y 163.058,Z 595.215,A -85,B 0,C 180,E1 -23390.072,E2 -23390.072} C_VEL
LIN {X 0,Y 165.114,Z 596.839,A -85,B 0,C 180,E1 -23395.116,E2 -23395.116} C_VEL
LIN {X 0,Y 168.677,Z 597.17,A -85,B 0,C 180,E1 -23400.548,E2 -23400.548} C_VEL
LIN {X 0,Y 172.468,Z 596.388,A -85,B 0,C 180,E1 -23404.674,E2 -23404.674} C_VEL
LIN {X 0,Y 177.994,Z 594.29,A -85,B 0,C 180,E1 -23409.214,E2 -23409.214} C_VEL
LIN {X 0,Y 184.199,Z 591.125,A -85,B 0,C 180,E1 -23413.233,E2 -23413.233} C_VEL
LIN {X 0,Y 191.676,Z 586.58,A -85,B 0,C 180,E1 -23417.057,E2 -23417.057} C_VEL
LIN {X 0,Y 200.001,Z 580.626,A -85,B 0,C 180,E1 -23420.573,E2 -23420.573} C_VEL
LIN {X 0,Y 209.237,Z 573.146,A -85,B 0,C 180,E1 -23423.77,E2 -23423.77} C_VEL
LIN {X 0,Y 215.379,Z 567.551,A -85,B 0,C 180,E1 -23425.617,E2 -23425.617} C_VEL
LIN {X 0,Y 216.174,Z 566.681,A -85,B 0,C 180,E1 -23426.033,E2 -23426.033} C_VEL
LIN {X 0,Y 216.54,Z 565.869,A -85,B 0,C 180,E1 -23427.025,E2 -23427.025} C_VEL
LIN {X 0,Y 216.888,Z 564.691,A -85,B 0,C 180,E1 -23429.082,E2 -23429.082} C_VEL
LIN {X 0,Y 217.073,Z 563.993,A -85,B 0,C 180,E1 -23431.199,E2 -23431.199} C_VEL
LIN {X 0,Y 216.979,Z 563.992,A -85,B 0,C 180,E1 -23433.41,E2 -23433.41} C_VEL
LIN {X 0,Y 216.65,Z 564.72,A -85,B 0,C 180,E1 -23435.809,E2 -23435.809} C_VEL
LIN {X 0,Y 216.06,Z 566.526,A -85,B 0,C 180,E1 -23438.679,E2 -23438.679} C_VEL
LIN {X 0,Y 215.069,Z 568.875,A -85,B 0,C 180,E1 -23440.81,E2 -23440.81} C_VEL
LIN {X 0,Y 211.985,Z 573.344,A -85,B 0,C 180,E1 -23443.167,E2 -23443.167} C_VEL
LIN {X 0,Y 208.792,Z 577.388,A -85,B 0,C 180,E1 -23445.02,E2 -23445.02} C_VEL
LIN {X 0,Y 207.342,Z 579.147,A -85,B 0,C 180,E1 -23445.762,E2 -23445.762} C_VEL
LIN {X 0,Y 200.094,Z 585.933,A -85,B 0,C 180,E1 -23448.138,E2 -23448.138} C_VEL
LIN {X 0,Y 191.394,Z 593.284,A -85,B 0,C 180,E1 -23451.374,E2 -23451.374} C_VEL
LIN {X 0,Y 185.688,Z 597.867,A -85,B 0,C 180,E1 -23454.081,E2 -23454.081} C_VEL
LIN {X 0,Y 178.882,Z 602.959,A -85,B 0,C 180,E1 -23457.969,E2 -23457.969} C_VEL
LIN {X 0,Y 174.485,Z 606.019,A -85,B 0,C 180,E1 -23461.097,E2 -23461.097} C_VEL
LIN {X 0,Y 168.7,Z 609.661,A -85,B 0,C 180,E1 -23466.421,E2 -23466.421} C_VEL
LIN {X 0,Y 165.912,Z 611.179,A -85,B 0,C 180,E1 -23470.192,E2 -23470.192} C_VEL
LIN {X 0,Y 163.463,Z 612.133,A -85,B 0,C 180,E1 -23475.051,E2 -23475.051} C_VEL
LIN {X 0,Y 162.361,Z 611.987,A -85,B 0,C 180,E1 -23480.029,E2 -23480.029} C_VEL
LIN {X 0,Y 162.295,Z 610.671,A -85,B 0,C 180,E1 -23485.032,E2 -23485.032} C_VEL
LIN {X 0,Y 162.724,Z 608.039,A -85,B 0,C 180,E1 -23490,E2 -23490} C_VEL
LIN {X 0,Y 162.649,Z 604.98,A -85,B 0,C 180,E1 -23493.716,E2 -23493.716} C_VEL
LIN {X 0,Y 162.718,Z 600.982,A -85,B 0,C 180,E1 -23497.445,E2 -23497.445} C_VEL
LIN {X 0,Y 163.287,Z 594.028,A -85,B 0,C 180,E1 -23502.427,E2 -23502.427} C_VEL
LIN {X 0,Y 164.439,Z 586.278,A -85,B 0,C 180,E1 -23506.767,E2 -23506.767} C_VEL
LIN {X 0,Y 166.508,Z 576.756,A -85,B 0,C 180,E1 -23511.024,E2 -23511.024} C_VEL
LIN {X 0,Y 167.107,Z 574.101,A -85,B 0,C 180,E1 -23512.044,E2 -23512.044} C_VEL
LIN {X 0,Y 167.493,Z 570.089,A -85,B 0,C 180,E1 -23513.519,E2 -23513.519} C_VEL
LIN {X 0,Y 166.709,Z 563.062,A -85,B 0,C 180,E1 -23515.883,E2 -23515.883} C_VEL
LIN {X 0,Y 165.606,Z 554.049,A -85,B 0,C 180,E1 -23518.565,E2 -23518.565} C_VEL
LIN {X 0,Y 165.697,Z 550.89,A -85,B 0,C 180,E1 -23519.4,E2 -23519.4} C_VEL
LIN {X 0,Y 165.192,Z 539.293,A -85,B 0,C 180,E1 -23522.266,E2 -23522.266} C_VEL
LIN {X 0,Y 164.389,Z 526.278,A -85,B 0,C 180,E1 -23525.022,E2 -23525.022} C_VEL
LIN {X 0,Y 163.195,Z 512.234,A -85,B 0,C 180,E1 -23527.552,E2 -23527.552} C_VEL
LIN {X 0,Y 161.618,Z 497.93,A -85,B 0,C 180,E1 -23529.723,E2 -23529.723} C_VEL
LIN {X 0,Y 159.882,Z 486.836,A -85,B 0,C 180,E1 -23531.17,E2 -23531.17} C_VEL
LIN {X 0,Y 159.194,Z 483.879,A -85,B 0,C 180,E1 -23531.573,E2 -23531.573} C_VEL
LIN {X 0,Y 158.852,Z 481.41,A -85,B 0,C 180,E1 -23535.062,E2 -23535.062} C_VEL
LIN {X 0,Y 158.245,Z 478.689,A -85,B 0,C 180,E1 -23539.025,E2 -23539.025} C_VEL
LIN {X 0,Y 157.522,Z 474.485,A -85,B 0,C 180,E1 -23545.524,E2 -23545.524} C_VEL
LIN {X 0,Y 157.286,Z 474.519,A -85,B 0,C 180,E1 -23550.561,E2 -23550.561} C_VEL
LIN {X 0,Y 157.32,Z 474.506,A -85,B 0,C 180,E1 -23553.466,E2 -23553.466} C_VEL
LIN {X 0,Y 157.394,Z 474.503,A -85,B 0,C 180,E1 -23559.666,E2 -23559.666} C_VEL
LIN {X 0,Y 157.483,Z 474.487,A -85,B 0,C 180,E1 -23564.469,E2 -23564.469} C_VEL
LIN {X 0,Y 157.732,Z 474.461,A -85,B 0,C 180,E1 -23569.734,E2 -23569.734} C_VEL
LIN {X 0,Y 157.807,Z 474.449,A -85,B 0,C 180,E1 -23572.322,E2 -23572.322} C_VEL
LIN {X 0,Y 158.255,Z 474.395,A -85,B 0,C 180,E1 -23580.001,E2 -23580.001} C_VEL
LIN {X 0,Y 157.807,Z 474.451,A -85,B 0,C 180,E1 -23587.679,E2 -23587.679} C_VEL
LIN {X 0,Y 157.681,Z 474.463,A -85,B 0,C 180,E1 -23591.32,E2 -23591.32} C_VEL
LIN {X 0,Y 157.46,Z 474.495,A -85,B 0,C 180,E1 -23595.534,E2 -23595.534} C_VEL
LIN {X 0,Y 157.369,Z 474.505,A -85,B 0,C 180,E1 -23600.934,E2 -23600.934} C_VEL
LIN {X 0,Y 157.314,Z 474.51,A -85,B 0,C 180,E1 -23606.685,E2 -23606.685} C_VEL
LIN {X 0,Y 157.278,Z 474.519,A -85,B 0,C 180,E1 -23612.428,E2 -23612.428} C_VEL
LIN {X 0,Y 157.282,Z 474.512,A -85,B 0,C 180,E1 -23616.458,E2 -23616.458} C_VEL
LIN {X 0,Y 157.213,Z 474.527,A -85,B 0,C 180,E1 -23622.111,E2 -23622.111} C_VEL
LIN {X 0,Y 157.215,Z 474.524,A -85,B 0,C 180,E1 -23627.892,E2 -23627.892} C_VEL
LIN {X 0,Y 157.284,Z 474.515,A -85,B 0,C 180,E1 -23633.544,E2 -23633.544} C_VEL
LIN {X 0,Y 157.296,Z 474.517,A -85,B 0,C 180,E1 -23638.096,E2 -23638.096} C_VEL
LIN {X 0,Y 157.324,Z 474.508,A -85,B 0,C 180,E1 -23643.467,E2 -23643.467} C_VEL
LIN {X 0,Y 157.397,Z 474.503,A -85,B 0,C 180,E1 -23649.668,E2 -23649.668} C_VEL
LIN {X 0,Y 157.457,Z 474.494,A -85,B 0,C 180,E1 -23654.466,E2 -23654.466} C_VEL
LIN {X 0,Y 157.69,Z 474.463,A -85,B 0,C 180,E1 -23659.731,E2 -23659.731} C_VEL
LIN {X 0,Y 157.766,Z 474.454,A -85,B 0,C 180,E1 -23662.32,E2 -23662.32} C_VEL
LIN {X 0,Y 158.26,Z 474.391,A -85,B 0,C 180,E1 -23670,E2 -23670} C_VEL
LIN {X 0,Y 157.774,Z 474.451,A -85,B 0,C 180,E1 -23677.68,E2 -23677.68} C_VEL
LIN {X 0,Y 157.641,Z 474.469,A -85,B 0,C 180,E1 -23681.238,E2 -23681.238} C_VEL
LIN {X 0,Y 157.464,Z 474.496,A -85,B 0,C 180,E1 -23685.533,E2 -23685.533} C_VEL
LIN {X 0,Y 157.374,Z 474.509,A -85,B 0,C 180,E1 -23690.932,E2 -23690.932} C_VEL
LIN {X 0,Y 157.313,Z 474.514,A -85,B 0,C 180,E1 -23696.681,E2 -23696.681} C_VEL
LIN {X 0,Y 157.271,Z 474.525,A -85,B 0,C 180,E1 -23701.294,E2 -23701.294} C_VEL
LIN {X 0,Y 162.2,Z 489.197,A -85,B 0,C 180,E1 -23703.908,E2 -23703.908} C_VEL
LIN {X 0,Y 166.207,Z 502.649,A -85,B 0,C 180,E1 -23706.602,E2 -23706.602} C_VEL
LIN {X 0,Y 168.842,Z 515.566,A -85,B 0,C 180,E1 -23709.403,E2 -23709.403} C_VEL
LIN {X 0,Y 169.445,Z 519.583,A -85,B 0,C 180,E1 -23710.341,E2 -23710.341} C_VEL
LIN {X 0,Y 166.577,Z 531.82,A -85,B 0,C 180,E1 -23713.058,E2 -23713.058} C_VEL
LIN {X 0,Y 163.736,Z 543.287,A -85,B 0,C 180,E1 -23716.2,E2 -23716.2} C_VEL
LIN {X 0,Y 160.923,Z 554.217,A -85,B 0,C 180,E1 -23719.895,E2 -23719.895} C_VEL
LIN {X 0,Y 158.498,Z 564.136,A -85,B 0,C 180,E1 -23724.064,E2 -23724.064} C_VEL
LIN {X 0,Y 156.852,Z 572.414,A -85,B 0,C 180,E1 -23728.354,E2 -23728.354} C_VEL
LIN {X 0,Y 155.519,Z 579.859,A -85,B 0,C 180,E1 -23733.133,E2 -23733.133} C_VEL
LIN {X 0,Y 154.928,Z 585.082,A -85,B 0,C 180,E1 -23737.319,E2 -23737.319} C_VEL
LIN {X 0,Y 154.721,Z 590.163,A -85,B 0,C 180,E1 -23742.531,E2 -23742.531} C_VEL
LIN {X 0,Y 155.169,Z 593.348,A -85,B 0,C 180,E1 -23746.911,E2 -23746.911} C_VEL
LIN {X 0,Y 156.696,Z 596.075,A -85,B 0,C 180,E1 -23752.267,E2 -23752.267} C_VEL
LIN {X 0,Y 159.256,Z 597.502,A -85,B 0,C 180,E1 -23757.47,E2 -23757.47} C_VEL
LIN {X 0,Y 162.93,Z 597.718,A -85,B 0,C 180,E1 -23762.472,E2 -23762.472} C_VEL
LIN {X 0,Y 167.801,Z 596.753,A -85,B 0,C 180,E1 -23767.218,E2 -23767.218} C_VEL
LIN {X 0,Y 173.811,Z 594.594,A -85,B 0,C 180,E1 -23771.664,E2 -23771.664} C_VEL
LIN {X 0,Y 180.89,Z 591.251,A -85,B 0,C 180,E1 -23775.781,E2 -23775.781} C_VEL
LIN {X 0,Y 188.999,Z 586.579,A -85,B 0,C 180,E1 -23779.552,E2 -23779.552} C_VEL
LIN {X 0,Y 198.072,Z 580.507,A -85,B 0,C 180,E1 -23782.973,E2 -23782.973} C_VEL
LIN {X 0,Y 207.857,Z 572.937,A -85,B 0,C 180,E1 -23786.075,E2 -23786.075} C_VEL
LIN {X 0,Y 210.397,Z 570.751,A -85,B 0,C 180,E1 -23786.804,E2 -23786.804} C_VEL
LIN {X 0,Y 211.05,Z 569.867,A -85,B 0,C 180,E1 -23787.788,E2 -23787.788} C_VEL
LIN {X 0,Y 211.482,Z 568.86,A -85,B 0,C 180,E1 -23790.229,E2 -23790.229} C_VEL
LIN {X 0,Y 211.643,Z 568.482,A -85,B 0,C 180,E1 -23792.094,E2 -23792.094} C_VEL
LIN {X 0,Y 211.362,Z 568.896,A -85,B 0,C 180,E1 -23794.42,E2 -23794.42} C_VEL
LIN {X 0,Y 210.914,Z 569.986,A -85,B 0,C 180,E1 -23796.898,E2 -23796.898} C_VEL
LIN {X 0,Y 209.996,Z 572.158,A -85,B 0,C 180,E1 -23799.67,E2 -23799.67} C_VEL
LIN {X 0,Y 209.444,Z 573.001,A -85,B 0,C 180,E1 -23800.287,E2 -23800.287} C_VEL
LIN {X 0,Y 206.457,Z 576.628,A -85,B 0,C 180,E1 -23802.309,E2 -23802.309} C_VEL
LIN {X 0,Y 202.836,Z 580.66,A -85,B 0,C 180,E1 -23804.236,E2 -23804.236} C_VEL
LIN {X 0,Y 199.739,Z 583.45,A -85,B 0,C 180,E1 -23805.275,E2 -23805.275} C_VEL
LIN {X 0,Y 190.382,Z 591.057,A -85,B 0,C 180,E1 -23808.359,E2 -23808.359} C_VEL
LIN {X 0,Y 181.861,Z 597.307,A -85,B 0,C 180,E1 -23811.807,E2 -23811.807} C_VEL
LIN {X 0,Y 174.621,Z 602.347,A -85,B 0,C 180,E1 -23815.705,E2 -23815.705} C_VEL
LIN {X 0,Y 168.285,Z 606.282,A -85,B 0,C 180,E1 -23819.924,E2 -23819.924} C_VEL
LIN {X 0,Y 163.093,Z 609.142,A -85,B 0,C 180,E1 -23824.474,E2 -23824.474} C_VEL
LIN {X 0,Y 159.207,Z 610.921,A -85,B 0,C 180,E1 -23829.32,E2 -23829.32} C_VEL
LIN {X 0,Y 156.572,Z 611.626,A -85,B 0,C 180,E1 -23834.377,E2 -23834.377} C_VEL
LIN {X 0,Y 155.368,Z 611.248,A -85,B 0,C 180,E1 -23839.576,E2 -23839.576} C_VEL
LIN {X 0,Y 155.253,Z 609.737,A -85,B 0,C 180,E1 -23844.806,E2 -23844.806} C_VEL
LIN {X 0,Y 155.42,Z 608.496,A -85,B 0,C 180,E1 -23847.408,E2 -23847.408} C_VEL
LIN {X 0,Y 155.695,Z 606.897,A -85,B 0,C 180,E1 -23850,E2 -23850} C_VEL
LIN {X 0,Y 155.641,Z 603.717,A -85,B 0,C 180,E1 -23853.884,E2 -23853.884} C_VEL
LIN {X 0,Y 155.702,Z 599.51,A -85,B 0,C 180,E1 -23857.782,E2 -23857.782} C_VEL
LIN {X 0,Y 156.369,Z 592.367,A -85,B 0,C 180,E1 -23862.986,E2 -23862.986} C_VEL
LIN {X 0,Y 157.639,Z 584.296,A -85,B 0,C 180,E1 -23867.513,E2 -23867.513} C_VEL
LIN {X 0,Y 159.816,Z 574.686,A -85,B 0,C 180,E1 -23871.824,E2 -23871.824} C_VEL
LIN {X 0,Y 162.169,Z 565.113,A -85,B 0,C 180,E1 -23875.303,E2 -23875.303} C_VEL
LIN {X 0,Y 165.082,Z 553.9,A -85,B 0,C 180,E1 -23878.616,E2 -23878.616} C_VEL
LIN {X 0,Y 165.697,Z 550.89,A -85,B 0,C 180,E1 -23879.4,E2 -23879.4} C_VEL
LIN {X 0,Y 165.56,Z 547.804,A -85,B 0,C 180,E1 -23880.21,E2 -23880.21} C_VEL
LIN {X 0,Y 164.765,Z 544.718,A -85,B 0,C 180,E1 -23881.023,E2 -23881.023} C_VEL
LIN {X 0,Y 162.056,Z 538.808,A -85,B 0,C 180,E1 -23882.632,E2 -23882.632} C_VEL
LIN {X 0,Y 158.493,Z 531.207,A -85,B 0,C 180,E1 -23884.62,E2 -23884.62} C_VEL
LIN {X 0,Y 157.427,Z 526.2,A -85,B 0,C 180,E1 -23885.746,E2 -23885.746} C_VEL
LIN {X 0,Y 156.279,Z 512.055,A -85,B 0,C 180,E1 -23888.41,E2 -23888.41} C_VEL
LIN {X 0,Y 154.79,Z 497.762,A -85,B 0,C 180,E1 -23890.667,E2 -23890.667} C_VEL
LIN {X 0,Y 153.174,Z 488.455,A -85,B 0,C 180,E1 -23891.976,E2 -23891.976} C_VEL
LIN {X 0,Y 152.083,Z 483.491,A -85,B 0,C 180,E1 -23892.683,E2 -23892.683} C_VEL
LIN {X 0,Y 151.34,Z 479.973,A -85,B 0,C 180,E1 -23897.988,E2 -23897.988} C_VEL
LIN {X 0,Y 150.498,Z 475.36,A -85,B 0,C 180,E1 -23905.412,E2 -23905.412} C_VEL
LIN {X 0,Y 150.244,Z 475.391,A -85,B 0,C 180,E1 -23912.717,E2 -23912.717} C_VEL
LIN {X 0,Y 150.35,Z 475.382,A -85,B 0,C 180,E1 -23919.207,E2 -23919.207} C_VEL
LIN {X 0,Y 150.388,Z 475.37,A -85,B 0,C 180,E1 -23923.717,E2 -23923.717} C_VEL
LIN {X 0,Y 150.656,Z 475.343,A -85,B 0,C 180,E1 -23929.246,E2 -23929.246} C_VEL
LIN {X 0,Y 150.742,Z 475.329,A -85,B 0,C 180,E1 -23931.96,E2 -23931.96} C_VEL
LIN {X 0,Y 151.216,Z 475.272,A -85,B 0,C 180,E1 -23940.001,E2 -23940.001} C_VEL
LIN {X 0,Y 150.743,Z 475.332,A -85,B 0,C 180,E1 -23948.041,E2 -23948.041} C_VEL
LIN {X 0,Y 150.612,Z 475.344,A -85,B 0,C 180,E1 -23951.506,E2 -23951.506} C_VEL
LIN {X 0,Y 150.366,Z 475.38,A -85,B 0,C 180,E1 -23956.287,E2 -23956.287} C_VEL
LIN {X 0,Y 150.35,Z 475.379,A -85,B 0,C 180,E1 -23960.793,E2 -23960.793} C_VEL
LIN {X 0,Y 150.243,Z 475.39,A -85,B 0,C 180,E1 -23967.283,E2 -23967.283} C_VEL
LIN {X 0,Y 150.218,Z 475.398,A -85,B 0,C 180,E1 -23972.635,E2 -23972.635} C_VEL
LIN {X 0,Y 150.211,Z 475.392,A -85,B 0,C 180,E1 -23977.463,E2 -23977.463} C_VEL
LIN {X 0,Y 150.154,Z 475.406,A -85,B 0,C 180,E1 -23981.507,E2 -23981.507} C_VEL
LIN {X 0,Y 150.143,Z 475.403,A -85,B 0,C 180,E1 -23985.403,E2 -23985.403} C_VEL
LIN {X 0,Y 150.159,Z 475.404,A -85,B 0,C 180,E1 -23989.062,E2 -23989.062} C_VEL
LIN {X 0,Y 150.217,Z 475.395,A -85,B 0,C 180,E1 -23992.69,E2 -23992.69} C_VEL
LIN {X 0,Y 150.22,Z 475.396,A -85,B 0,C 180,E1 -23997.366,E2 -23997.366} C_VEL
LIN {X 0,Y 150.246,Z 475.389,A -85,B 0,C 180,E1 -24002.718,E2 -24002.718} C_VEL
LIN {X 0,Y 150.354,Z 475.381,A -85,B 0,C 180,E1 -24009.208,E2 -24009.208} C_VEL
LIN {X 0,Y 150.364,Z 475.377,A -85,B 0,C 180,E1 -24013.714,E2 -24013.714} C_VEL
LIN {X 0,Y 150.613,Z 475.347,A -85,B 0,C 180,E1 -24019.243,E2 -24019.243} C_VEL
LIN {X 0,Y 150.704,Z 475.334,A -85,B 0,C 180,E1 -24021.958,E2 -24021.958} C_VEL
LIN {X 0,Y 151.221,Z 475.267,A -85,B 0,C 180,E1 -24030,E2 -24030} C_VEL
LIN {X 0,Y 150.711,Z 475.33,A -85,B 0,C 180,E1 -24038.042,E2 -24038.042} C_VEL
LIN {X 0,Y 150.581,Z 475.349,A -85,B 0,C 180,E1 -24041.439,E2 -24041.439} C_VEL
LIN {X 0,Y 150.372,Z 475.379,A -85,B 0,C 180,E1 -24046.285,E2 -24046.285} C_VEL
LIN {X 0,Y 150.355,Z 475.383,A -85,B 0,C 180,E1 -24050.793,E2 -24050.793} C_VEL
LIN {X 0,Y 150.235,Z 475.398,A -85,B 0,C 180,E1 -24057.273,E2 -24057.273} C_VEL
LIN {X 0,Y 150.249,Z 475.604,A -85,B 0,C 180,E1 -24060.284,E2 -24060.284} C_VEL
LIN {X 0,Y 155.038,Z 489.491,A -85,B 0,C 180,E1 -24062.954,E2 -24062.954} C_VEL
LIN {X 0,Y 159.016,Z 502.87,A -85,B 0,C 180,E1 -24065.748,E2 -24065.748} C_VEL
LIN {X 0,Y 160.972,Z 511.527,A -85,B 0,C 180,E1 -24067.678,E2 -24067.678} C_VEL
LIN {X 0,Y 162.449,Z 520.637,A -85,B 0,C 180,E1 -24069.849,E2 -24069.849} C_VEL
LIN {X 0,Y 159.303,Z 533.288,A -85,B 0,C 180,E1 -24072.823,E2 -24072.823} C_VEL
LIN {X 0,Y 156.42,Z 544.508,A -85,B 0,C 180,E1 -24076.112,E2 -24076.112} C_VEL
LIN {X 0,Y 153.499,Z 555.624,A -85,B 0,C 180,E1 -24080.133,E2 -24080.133} C_VEL
LIN {X 0,Y 151.152,Z 565.302,A -85,B 0,C 180,E1 -24084.464,E2 -24084.464} C_VEL
LIN {X 0,Y 149.57,Z 573.321,A -85,B 0,C 180,E1 -24088.877,E2 -24088.877} C_VEL
LIN {X 0,Y 148.415,Z 579.716,A -85,B 0,C 180,E1 -24093.181,E2 -24093.181} C_VEL
LIN {X 0,Y 147.794,Z 585.089,A -85,B 0,C 180,E1 -24097.639,E2 -24097.639} C_VEL
LIN {X 0,Y 147.667,Z 590.519,A -85,B 0,C 180,E1 -24103.407,E2 -24103.407} C_VEL
LIN {X 0,Y 148.523,Z 594.402,A -85,B 0,C 180,E1 -24109.089,E2 -24109.089} C_VEL
LIN {X 0,Y 150.508,Z 596.908,A -85,B 0,C 180,E1 -24114.641,E2 -24114.641} C_VEL
LIN {X 0,Y 153.648,Z 598.172,A -85,B 0,C 180,E1 -24119.999,E2 -24119.999} C_VEL
LIN {X 0,Y 157.948,Z 598.243,A -85,B 0,C 180,E1 -24125.105,E2 -24125.105} C_VEL
LIN {X 0,Y 164.398,Z 596.923,A -85,B 0,C 180,E1 -24130.507,E2 -24130.507} C_VEL
LIN {X 0,Y 170.248,Z 594.882,A -85,B 0,C 180,E1 -24134.34,E2 -24134.34} C_VEL
LIN {X 0,Y 178.036,Z 591.408,A -85,B 0,C 180,E1 -24138.409,E2 -24138.409} C_VEL
LIN {X 0,Y 186.798,Z 586.659,A -85,B 0,C 180,E1 -24142.1,E2 -24142.1} C_VEL
LIN {X 0,Y 196.508,Z 580.495,A -85,B 0,C 180,E1 -24145.415,E2 -24145.415} C_VEL
LIN {X 0,Y 204.203,Z 574.843,A -85,B 0,C 180,E1 -24147.686,E2 -24147.686} C_VEL
LIN {X 0,Y 205.45,Z 573.753,A -85,B 0,C 180,E1 -24148.614,E2 -24148.614} C_VEL
LIN {X 0,Y 205.94,Z 572.938,A -85,B 0,C 180,E1 -24151.444,E2 -24151.444} C_VEL
LIN {X 0,Y 205.956,Z 572.979,A -85,B 0,C 180,E1 -24153.091,E2 -24153.091} C_VEL
LIN {X 0,Y 205.476,Z 573.748,A -85,B 0,C 180,E1 -24155.553,E2 -24155.553} C_VEL
LIN {X 0,Y 204.428,Z 575.948,A -85,B 0,C 180,E1 -24159.053,E2 -24159.053} C_VEL
LIN {X 0,Y 202.729,Z 577.865,A -85,B 0,C 180,E1 -24160.301,E2 -24160.301} C_VEL
LIN {X 0,Y 199.306,Z 581.368,A -85,B 0,C 180,E1 -24162.226,E2 -24162.226} C_VEL
LIN {X 0,Y 197.327,Z 583.195,A -85,B 0,C 180,E1 -24163.104,E2 -24163.104} C_VEL
LIN {X 0,Y 187.566,Z 590.627,A -85,B 0,C 180,E1 -24166.118,E2 -24166.118} C_VEL
LIN {X 0,Y 180.642,Z 595.433,A -85,B 0,C 180,E1 -24168.594,E2 -24168.594} C_VEL
LIN {X 0,Y 174.456,Z 599.438,A -85,B 0,C 180,E1 -24171.361,E2 -24171.361} C_VEL
LIN {X 0,Y 165.34,Z 604.801,A -85,B 0,C 180,E1 -24176.456,E2 -24176.456} C_VEL
LIN {X 0,Y 159.258,Z 607.882,A -85,B 0,C 180,E1 -24180.96,E2 -24180.96} C_VEL
LIN {X 0,Y 154.426,Z 609.943,A -85,B 0,C 180,E1 -24185.821,E2 -24185.821} C_VEL
LIN {X 0,Y 150.985,Z 610.973,A -85,B 0,C 180,E1 -24190.984,E2 -24190.984} C_VEL
LIN {X 0,Y 148.866,Z 610.937,A -85,B 0,C 180,E1 -24196.347,E2 -24196.347} C_VEL
LIN {X 0,Y 148.16,Z 609.786,A -85,B 0,C 180,E1 -24201.819,E2 -24201.819} C_VEL
LIN {X 0,Y 148.238,Z 608.744,A -85,B 0,C 180,E1 -24204.629,E2 -24204.629} C_VEL
LIN {X 0,Y 148.686,Z 605.751,A -85,B 0,C 180,E1 -24210,E2 -24210} C_VEL
LIN {X 0,Y 148.633,Z 602.348,A -85,B 0,C 180,E1 -24214.067,E2 -24214.067} C_VEL
LIN {X 0,Y 148.687,Z 597.985,A -85,B 0,C 180,E1 -24218.152,E2 -24218.152} C_VEL
LIN {X 0,Y 149.328,Z 591.541,A -85,B 0,C 180,E1 -24222.918,E2 -24222.918} C_VEL
LIN {X 0,Y 150.625,Z 583.46,A -85,B 0,C 180,E1 -24227.655,E2 -24227.655} C_VEL
LIN {X 0,Y 152.824,Z 573.857,A -85,B 0,C 180,E1 -24232.162,E2 -24232.162} C_VEL
LIN {X 0,Y 155.202,Z 564.433,A -85,B 0,C 180,E1 -24235.731,E2 -24235.731} C_VEL
LIN {X 0,Y 158.268,Z 552.972,A -85,B 0,C 180,E1 -24239.239,E2 -24239.239} C_VEL
LIN {X 0,Y 158.698,Z 550.602,A -85,B 0,C 180,E1 -24239.881,E2 -24239.881} C_VEL
LIN {X 0,Y 158.172,Z 538.652,A -85,B 0,C 180,E1 -24242.975,E2 -24242.975} C_VEL
LIN {X 0,Y 157.427,Z 526.2,A -85,B 0,C 180,E1 -24245.746,E2 -24245.746} C_VEL
LIN {X 0,Y 156.447,Z 521.175,A -85,B 0,C 180,E1 -24246.821,E2 -24246.821} C_VEL
LIN {X 0,Y 152.965,Z 513.251,A -85,B 0,C 180,E1 -24248.621,E2 -24248.621} C_VEL
LIN {X 0,Y 149.41,Z 505.174,A -85,B 0,C 180,E1 -24250.37,E2 -24250.37} C_VEL
LIN {X 0,Y 148.196,Z 499.899,A -85,B 0,C 180,E1 -24251.307,E2 -24251.307} C_VEL
LIN {X 0,Y 146.844,Z 491.017,A -85,B 0,C 180,E1 -24252.684,E2 -24252.684} C_VEL
LIN {X 0,Y 144.84,Z 483.087,A -85,B 0,C 180,E1 -24253.926,E2 -24253.926} C_VEL
LIN {X 0,Y 144.11,Z 480.002,A -85,B 0,C 180,E1 -24258.825,E2 -24258.825} C_VEL
LIN {X 0,Y 143.468,Z 476.236,A -85,B 0,C 180,E1 -24265.369,E2 -24265.369} C_VEL
LIN {X 0,Y 143.192,Z 476.272,A -85,B 0,C 180,E1 -24272.06,E2 -24272.06} C_VEL
LIN {X 0,Y 143.276,Z 476.263,A -85,B 0,C 180,E1 -24278.745,E2 -24278.745} C_VEL
LIN {X 0,Y 143.32,Z 476.253,A -85,B 0,C 180,E1 -24282.89,E2 -24282.89} C_VEL
LIN {X 0,Y 143.592,Z 476.225,A -85,B 0,C 180,E1 -24288.71,E2 -24288.71} C_VEL
LIN {X 0,Y 143.663,Z 476.21,A -85,B 0,C 180,E1 -24291.561,E2 -24291.561} C_VEL
LIN {X 0,Y 144.175,Z 476.149,A -85,B 0,C 180,E1 -24300.001,E2 -24300.001} C_VEL
LIN {X 0,Y 143.664,Z 476.213,A -85,B 0,C 180,E1 -24308.44,E2 -24308.44} C_VEL
LIN {X 0,Y 143.547,Z 476.224,A -85,B 0,C 180,E1 -24311.713,E2 -24311.713} C_VEL
LIN {X 0,Y 143.304,Z 476.257,A -85,B 0,C 180,E1 -24317.114,E2 -24317.114} C_VEL
LIN {X 0,Y 143.276,Z 476.26,A -85,B 0,C 180,E1 -24321.255,E2 -24321.255} C_VEL
LIN {X 0,Y 143.19,Z 476.268,A -85,B 0,C 180,E1 -24327.938,E2 -24327.938} C_VEL
LIN {X 0,Y 143.168,Z 476.276,A -85,B 0,C 180,E1 -24333.436,E2 -24333.436} C_VEL
LIN {X 0,Y 143.075,Z 476.286,A -85,B 0,C 180,E1 -24339.686,E2 -24339.686} C_VEL
LIN {X 0,Y 143.063,Z 476.288,A -85,B 0,C 180,E1 -24343.454,E2 -24343.454} C_VEL
LIN {X 0,Y 143.073,Z 476.284,A -85,B 0,C 180,E1 -24347.463,E2 -24347.463} C_VEL
LIN {X 0,Y 143.109,Z 476.284,A -85,B 0,C 180,E1 -24351.791,E2 -24351.791} C_VEL
LIN {X 0,Y 143.187,Z 476.272,A -85,B 0,C 180,E1 -24357.323,E2 -24357.323} C_VEL
LIN {X 0,Y 143.193,Z 476.269,A -85,B 0,C 180,E1 -24362.063,E2 -24362.063} C_VEL
LIN {X 0,Y 143.279,Z 476.261,A -85,B 0,C 180,E1 -24368.746,E2 -24368.746} C_VEL
LIN {X 0,Y 143.304,Z 476.253,A -85,B 0,C 180,E1 -24372.887,E2 -24372.887} C_VEL
LIN {X 0,Y 143.539,Z 476.228,A -85,B 0,C 180,E1 -24378.706,E2 -24378.706} C_VEL
LIN {X 0,Y 143.626,Z 476.214,A -85,B 0,C 180,E1 -24381.559,E2 -24381.559} C_VEL
LIN {X 0,Y 144.179,Z 476.144,A -85,B 0,C 180,E1 -24390,E2 -24390} C_VEL
LIN {X 0,Y 143.631,Z 476.212,A -85,B 0,C 180,E1 -24398.441,E2 -24398.441} C_VEL
LIN {X 0,Y 143.509,Z 476.231,A -85,B 0,C 180,E1 -24401.632,E2 -24401.632} C_VEL
LIN {X 0,Y 143.311,Z 476.256,A -85,B 0,C 180,E1 -24407.112,E2 -24407.112} C_VEL
LIN {X 0,Y 143.28,Z 476.263,A -85,B 0,C 180,E1 -24411.255,E2 -24411.255} C_VEL
LIN {X 0,Y 143.183,Z 476.276,A -85,B 0,C 180,E1 -24417.929,E2 -24417.929} C_VEL
LIN {X 0,Y 143.173,Z 476.281,A -85,B 0,C 180,E1 -24419.155,E2 -24419.155} C_VEL
LIN {X 0,Y 147.914,Z 489.8,A -85,B 0,C 180,E1 -24421.91,E2 -24421.91} C_VEL
